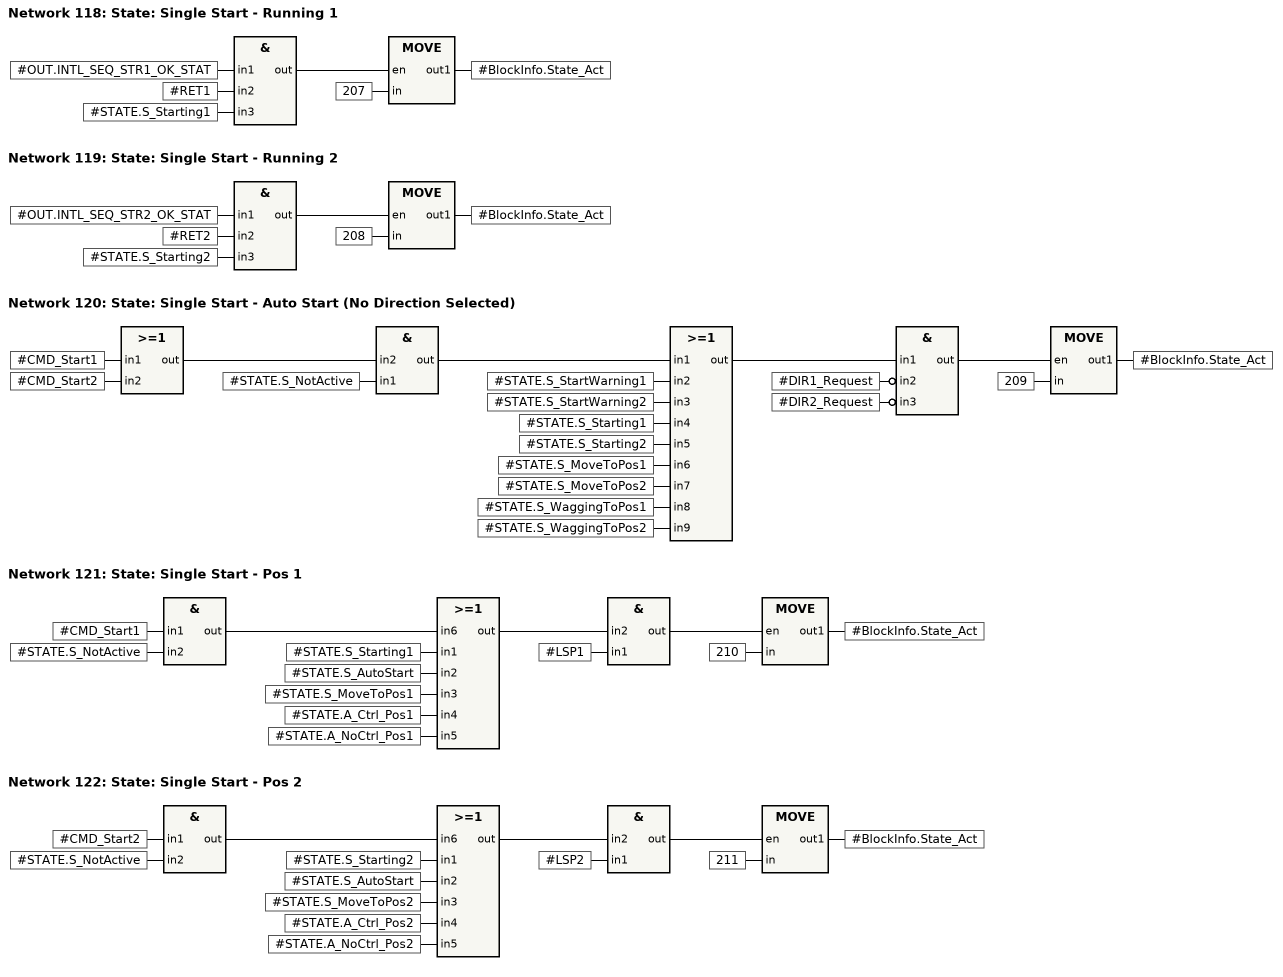
   IF #OUT.INTL_SEQ_STR1_OK_STAT AND #RET1 AND #STATE.S_Starting1 THEN #BlockInfo.State_Act := 207; END_IF;
END_REGION

REGION Network 119: State: Single Start - Running 2
   IF #OUT.INTL_SEQ_STR2_OK_STAT AND #RET2 AND #STATE.S_Starting2 THEN #BlockInfo.State_Act := 208; END_IF;
END_REGION

REGION Network 120: State: Single Start - Auto Start (No Direction Selected)
   IF (((#CMD_Start1 OR #CMD_Start2) AND #STATE.S_NotActive) OR #STATE.S_StartWarning1 OR #STATE.S_StartWarning2 OR #STATE.S_Starting1 OR #STATE.S_Starting2 OR #STATE.S_MoveToPos1 OR #STATE.S_MoveToPos2 OR #STATE.S_WaggingToPos1 OR #STATE.S_WaggingToPos2) AND NOT #DIR1_Request AND NOT #DIR2_Request THEN
       #BlockInfo.State_Act := 209;
   END_IF;
END_REGION

REGION Network 121: State: Single Start - Pos 1
   IF ((#CMD_Start1 AND #STATE.S_NotActive) OR #STATE.S_Starting1 OR #STATE.S_AutoStart OR #STATE.S_MoveToPos1 OR #STATE.A_Ctrl_Pos1 OR #STATE.A_NoCtrl_Pos1) AND #LSP1 THEN
       #BlockInfo.State_Act := 210;
   END_IF;
END_REGION

REGION Network 122: State: Single Start - Pos 2
   IF ((#CMD_Start2 AND #STATE.S_NotActive) OR #STATE.S_Starting2 OR #STATE.S_AutoStart OR #STATE.S_MoveToPos2 OR #STATE.A_Ctrl_Pos2 OR #STATE.A_NoCtrl_Pos2) AND #LSP2 THEN
       #BlockInfo.State_Act := 211;
   END_IF;
END_REGION

REGION Network 123: State: Single Start - Stop
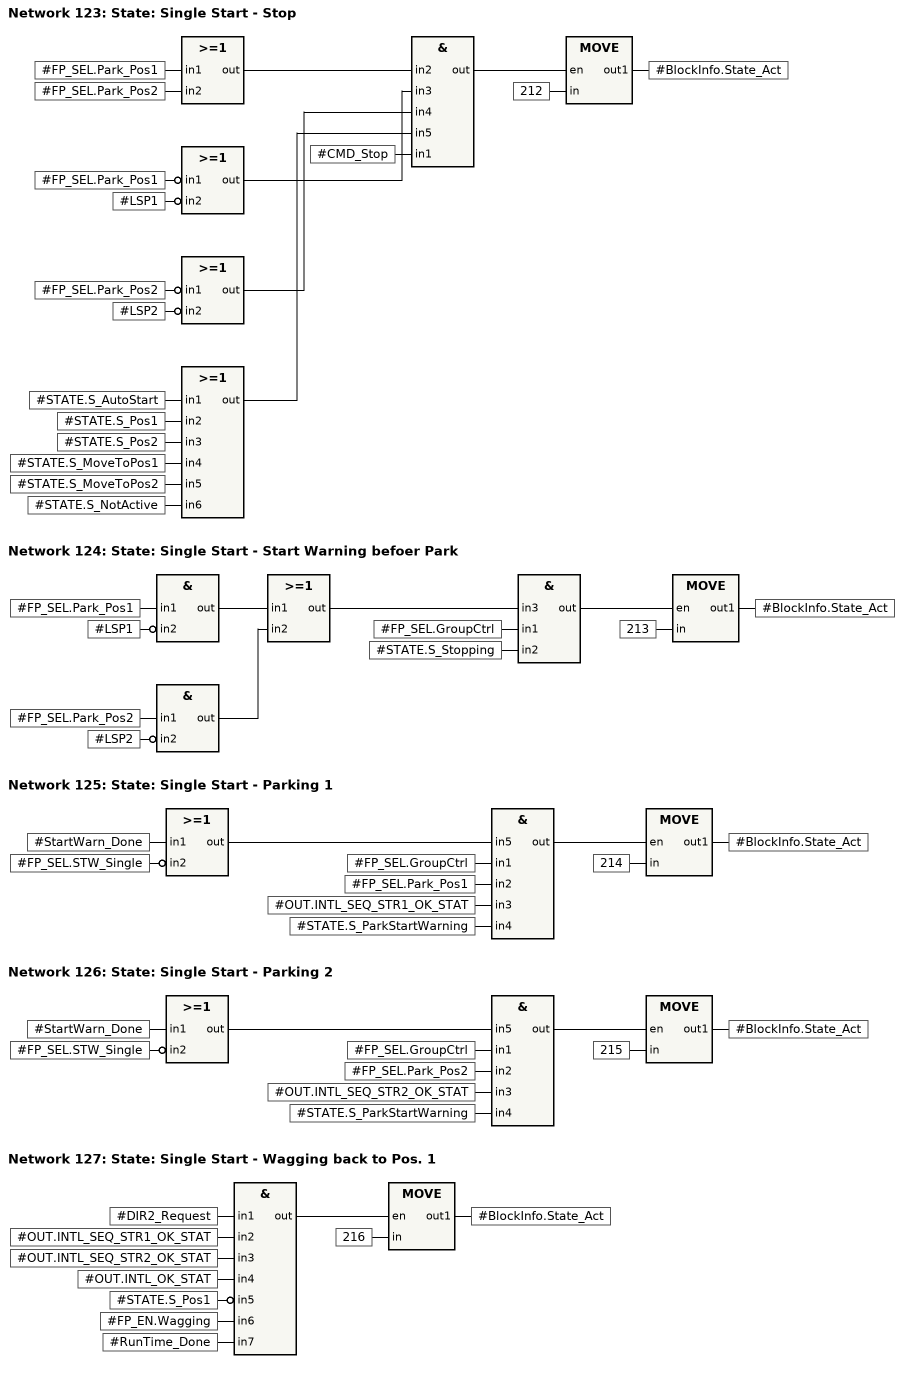
   IF (#FP_SEL.Park_Pos1 OR #FP_SEL.Park_Pos2) AND (NOT #FP_SEL.Park_Pos1 OR NOT #LSP1) AND (NOT #FP_SEL.Park_Pos2 OR NOT #LSP2) AND (#STATE.S_AutoStart OR #STATE.S_Pos1 OR #STATE.S_Pos2 OR #STATE.S_MoveToPos1 OR #STATE.S_MoveToPos2 OR #STATE.S_NotActive) AND #CMD_Stop THEN
       #BlockInfo.State_Act := 212;
   END_IF;
END_REGION

REGION Network 124: State: Single Start - Start Warning befoer Park
   IF ((#FP_SEL.Park_Pos1 AND NOT #LSP1) OR (#FP_SEL.Park_Pos2 AND NOT #LSP2)) AND #FP_SEL.GroupCtrl AND #STATE.S_Stopping THEN
       #BlockInfo.State_Act := 213;
   END_IF;
END_REGION

REGION Network 125: State: Single Start - Parking 1
   IF (#StartWarn_Done OR NOT #FP_SEL.STW_Single) AND #FP_SEL.GroupCtrl AND #FP_SEL.Park_Pos1 AND #OUT.INTL_SEQ_STR1_OK_STAT AND #STATE.S_ParkStartWarning THEN
       #BlockInfo.State_Act := 214;
   END_IF;
END_REGION

REGION Network 126: State: Single Start - Parking 2
   IF (#StartWarn_Done OR NOT #FP_SEL.STW_Single) AND #FP_SEL.GroupCtrl AND #FP_SEL.Park_Pos2 AND #OUT.INTL_SEQ_STR2_OK_STAT AND #STATE.S_ParkStartWarning THEN
       #BlockInfo.State_Act := 215;
   END_IF;
END_REGION

REGION Network 127: State: Single Start - Wagging back to Pos. 1
   IF #DIR2_Request AND #OUT.INTL_SEQ_STR1_OK_STAT AND #OUT.INTL_SEQ_STR2_OK_STAT AND #OUT.INTL_OK_STAT AND NOT #STATE.S_Pos1 AND #FP_EN.Wagging AND #RunTime_Done THEN
       #BlockInfo.State_Act := 216;
   END_IF;
END_REGION

REGION Network 128: State: Single Start - Wagging back to Pos. 2
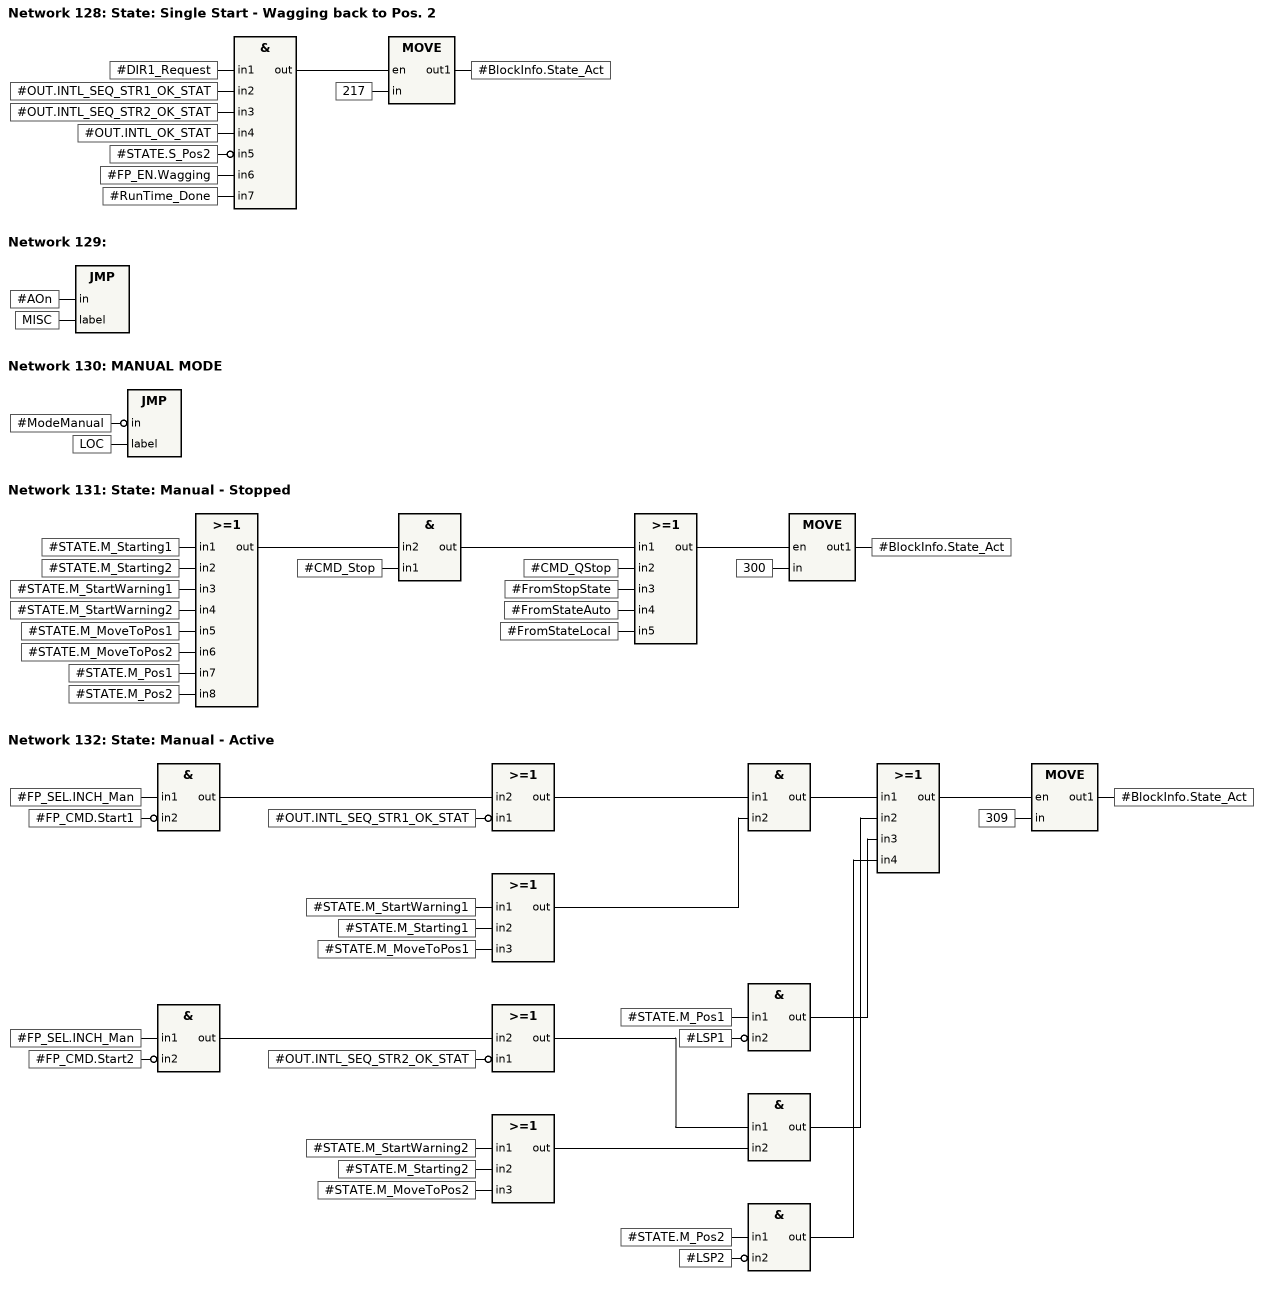
   IF #DIR1_Request AND #OUT.INTL_SEQ_STR1_OK_STAT AND #OUT.INTL_SEQ_STR2_OK_STAT AND #OUT.INTL_OK_STAT AND NOT #STATE.S_Pos2 AND #FP_EN.Wagging AND #RunTime_Done THEN
       #BlockInfo.State_Act := 217;
   END_IF;
END_REGION

REGION Network 129
   IF #AOn THEN GOTO MISC; END_IF;
END_REGION

REGION Network 130: MANUAL MODE
   MAN:
   IF NOT #ModeManual THEN GOTO LOC; END_IF;
END_REGION

REGION Network 131: State: Manual - Stopped
   IF ((#STATE.M_Starting1 OR #STATE.M_Starting2 OR #STATE.M_StartWarning1 OR #STATE.M_StartWarning2 OR #STATE.M_MoveToPos1 OR #STATE.M_MoveToPos2 OR #STATE.M_Pos1 OR #STATE.M_Pos2) AND #CMD_Stop) OR #CMD_QStop OR #FromStopState OR #FromStateAuto OR #FromStateLocal THEN
       #BlockInfo.State_Act := 300;
   END_IF;
END_REGION

REGION Network 132: State: Manual - Active
   // Build 016 - 21.Feb.2022 (SURAM-IN) FP_CMD.Start1,  FP_CMD.Start2 and FP_SEL.INCH_Man logic added for Inching in Manual Mode
   IF (((#FP_SEL.INCH_Man AND NOT #FP_CMD.Start1) OR NOT #OUT.INTL_SEQ_STR1_OK_STAT) AND (#STATE.M_StartWarning1 OR #STATE.M_Starting1 OR #STATE.M_MoveToPos1)) OR (((#FP_SEL.INCH_Man AND NOT #FP_CMD.Start2) OR NOT #OUT.INTL_SEQ_STR2_OK_STAT) AND (#STATE.M_StartWarning2 OR #STATE.M_Starting2 OR #STATE.M_MoveToPos2)) OR (#STATE.M_Pos1 AND NOT #LSP1) OR (#STATE.M_Pos2 AND NOT #LSP2) THEN
       #BlockInfo.State_Act := 309;
   END_IF;
END_REGION

REGION Network 133: State: Manual - Start Warning 1
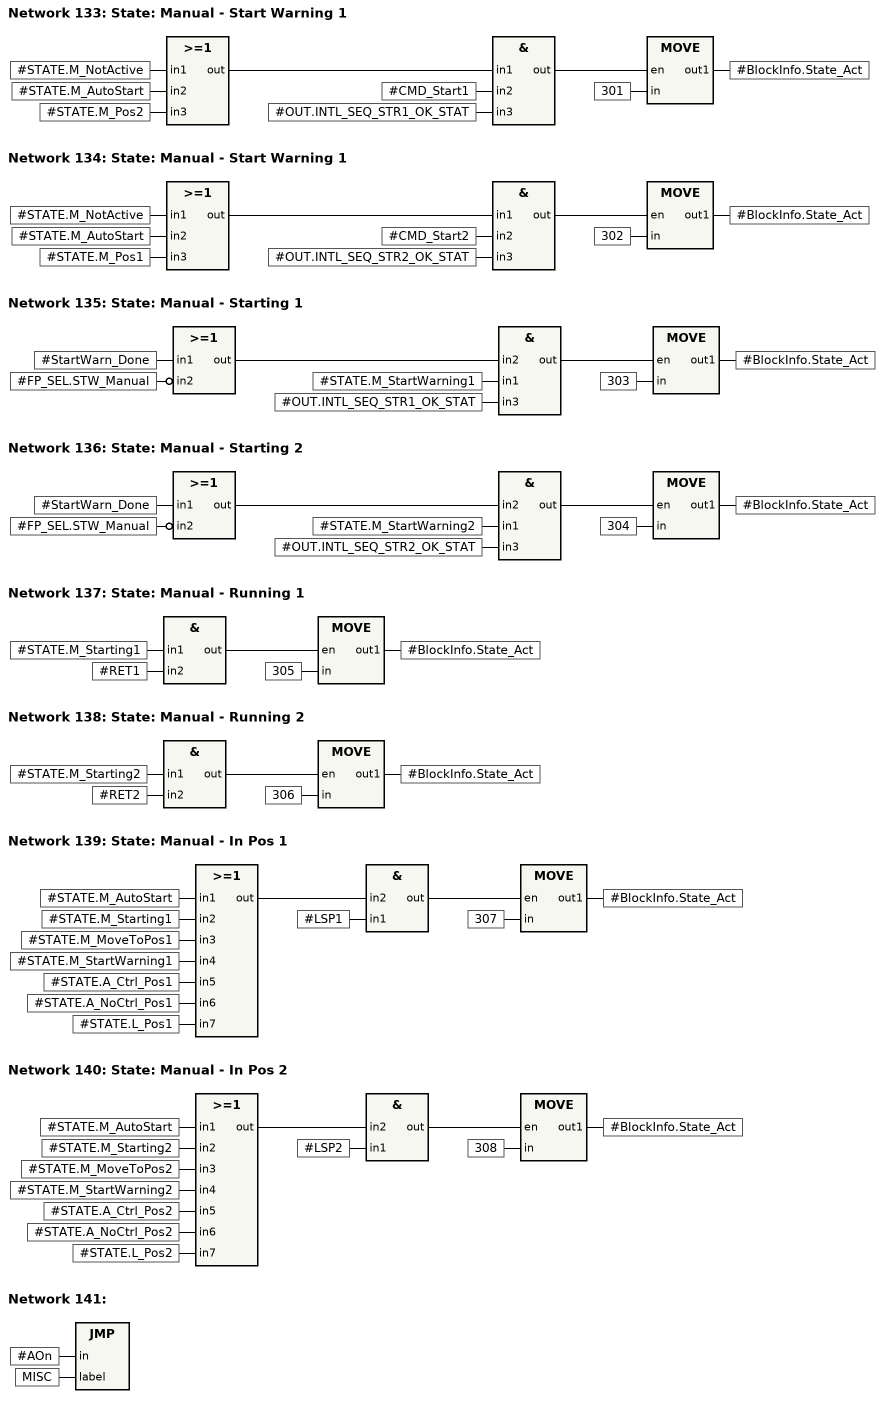
   IF (#STATE.M_NotActive OR #STATE.M_AutoStart OR #STATE.M_Pos2) AND #CMD_Start1 AND #OUT.INTL_SEQ_STR1_OK_STAT THEN
       #BlockInfo.State_Act := 301;
   END_IF;
END_REGION

REGION Network 134: State: Manual - Start Warning 1
   IF (#STATE.M_NotActive OR #STATE.M_AutoStart OR #STATE.M_Pos1) AND #CMD_Start2 AND #OUT.INTL_SEQ_STR2_OK_STAT THEN
       #BlockInfo.State_Act := 302;
   END_IF;
END_REGION

REGION Network 135: State: Manual - Starting 1
   IF (#StartWarn_Done OR NOT #FP_SEL.STW_Manual) AND #STATE.M_StartWarning1 AND #OUT.INTL_SEQ_STR1_OK_STAT THEN
       #BlockInfo.State_Act := 303;
   END_IF;
END_REGION

REGION Network 136: State: Manual - Starting 2
   IF (#StartWarn_Done OR NOT #FP_SEL.STW_Manual) AND #STATE.M_StartWarning2 AND #OUT.INTL_SEQ_STR2_OK_STAT THEN
       #BlockInfo.State_Act := 304;
   END_IF;
END_REGION

REGION Network 137: State: Manual - Running 1
   IF #STATE.M_Starting1 AND #RET1 THEN #BlockInfo.State_Act := 305; END_IF;
END_REGION

REGION Network 138: State: Manual - Running 2
   IF #STATE.M_Starting2 AND #RET2 THEN #BlockInfo.State_Act := 306; END_IF;
END_REGION

REGION Network 139: State: Manual - In Pos 1
   IF (#STATE.M_AutoStart OR #STATE.M_Starting1 OR #STATE.M_MoveToPos1 OR #STATE.M_StartWarning1 OR #STATE.A_Ctrl_Pos1 OR #STATE.A_NoCtrl_Pos1 OR #STATE.L_Pos1) AND #LSP1 THEN
       #BlockInfo.State_Act := 307;
   END_IF;
END_REGION

REGION Network 140: State: Manual - In Pos 2
   IF (#STATE.M_AutoStart OR #STATE.M_Starting2 OR #STATE.M_MoveToPos2 OR #STATE.M_StartWarning2 OR #STATE.A_Ctrl_Pos2 OR #STATE.A_NoCtrl_Pos2 OR #STATE.L_Pos2) AND #LSP2 THEN
       #BlockInfo.State_Act := 308;
   END_IF;
END_REGION

REGION Network 141
   IF #AOn THEN GOTO MISC; END_IF;
END_REGION

REGION Network 142: LOCAL MODE
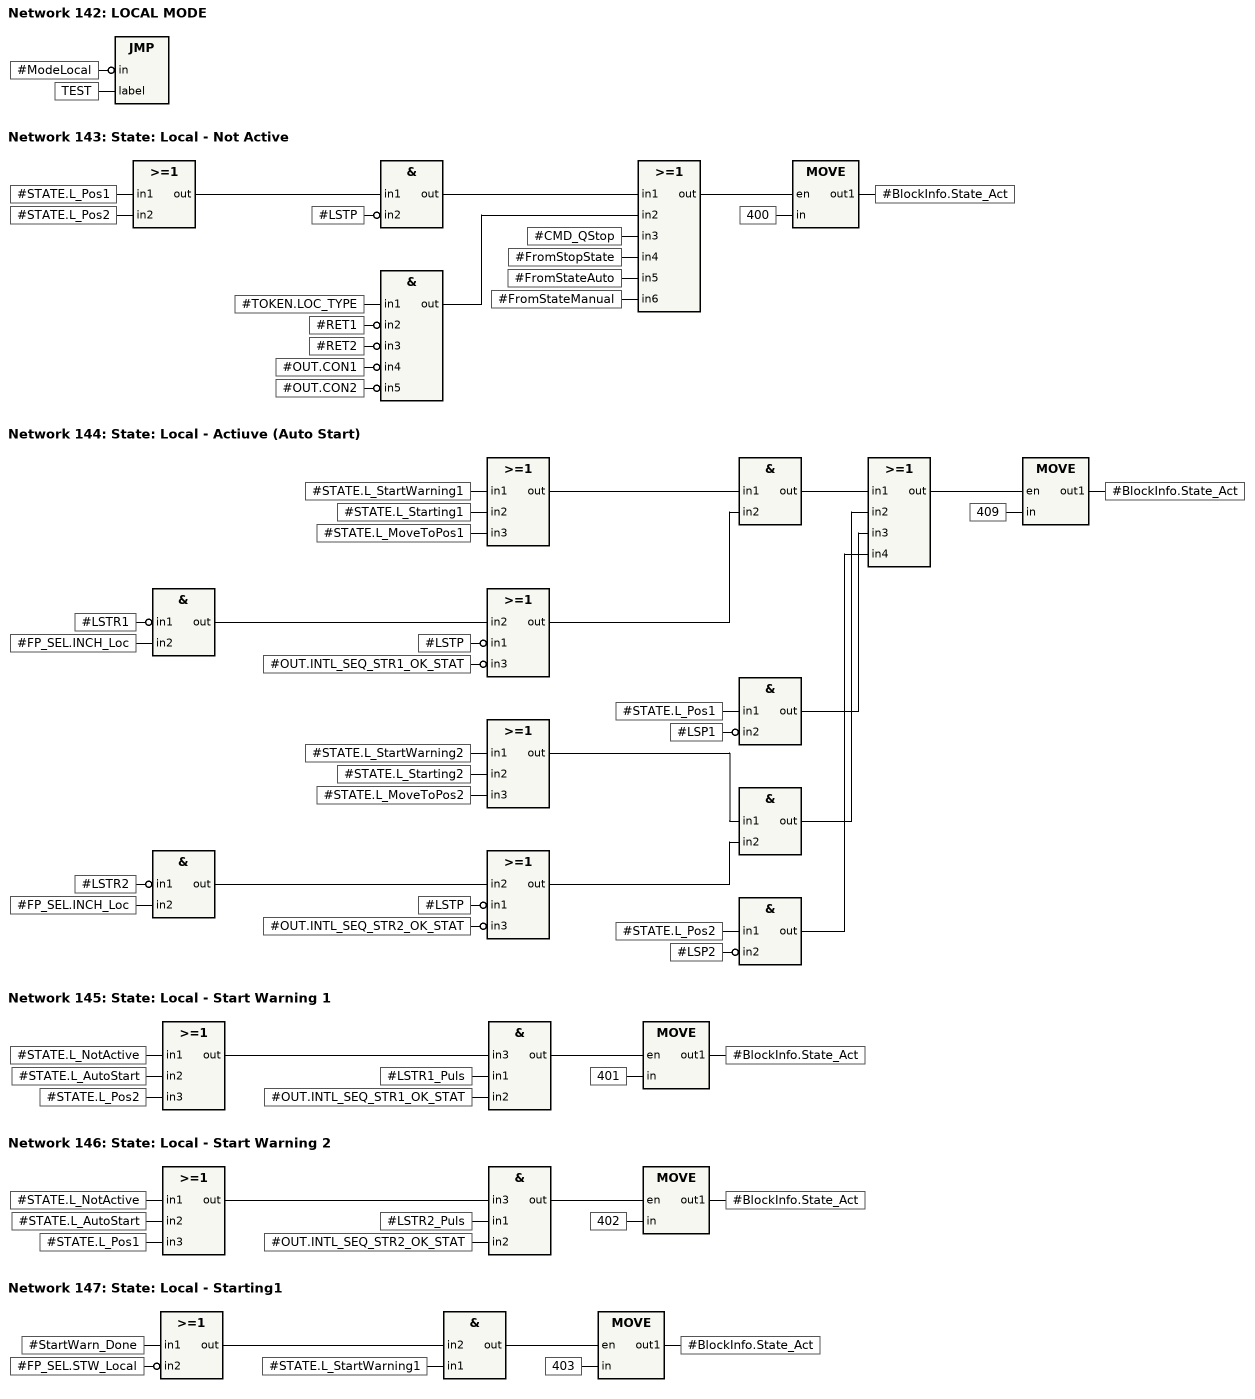
   LOC:
   IF NOT #ModeLocal THEN GOTO TEST; END_IF;
END_REGION

REGION Network 143: State: Local - Not Active
   IF ((#STATE.L_Pos1 OR #STATE.L_Pos2) AND NOT #LSTP) OR (#TOKEN.LOC_TYPE AND NOT #RET1 AND NOT #RET2 AND NOT #OUT.CON1 AND NOT #OUT.CON2) OR #CMD_QStop OR #FromStopState OR #FromStateAuto OR #FromStateManual THEN
       #BlockInfo.State_Act := 400;
   END_IF;
END_REGION

REGION Network 144: State: Local - Actiuve (Auto Start)
   IF ((#STATE.L_StartWarning1 OR #STATE.L_Starting1 OR #STATE.L_MoveToPos1) AND ((NOT #LSTR1 AND #FP_SEL.INCH_Loc) OR NOT #LSTP OR NOT #OUT.INTL_SEQ_STR1_OK_STAT)) OR ((#STATE.L_StartWarning2 OR #STATE.L_Starting2 OR #STATE.L_MoveToPos2) AND ((NOT #LSTR2 AND #FP_SEL.INCH_Loc) OR NOT #LSTP OR NOT #OUT.INTL_SEQ_STR2_OK_STAT)) OR (#STATE.L_Pos1 AND NOT #LSP1) OR (#STATE.L_Pos2 AND NOT #LSP2) THEN
       #BlockInfo.State_Act := 409;
   END_IF;
END_REGION

REGION Network 145: State: Local - Start Warning 1
   IF (#STATE.L_NotActive OR #STATE.L_AutoStart OR #STATE.L_Pos2) AND #LSTR1_Puls AND #OUT.INTL_SEQ_STR1_OK_STAT THEN
       #BlockInfo.State_Act := 401;
   END_IF;
END_REGION

REGION Network 146: State: Local - Start Warning 2
   IF (#STATE.L_NotActive OR #STATE.L_AutoStart OR #STATE.L_Pos1) AND #LSTR2_Puls AND #OUT.INTL_SEQ_STR2_OK_STAT THEN
       #BlockInfo.State_Act := 402;
   END_IF;
END_REGION

REGION Network 147: State: Local - Starting1
   IF (#StartWarn_Done OR NOT #FP_SEL.STW_Local) AND #STATE.L_StartWarning1 THEN
       #BlockInfo.State_Act := 403;
   END_IF;
END_REGION

REGION Network 148: State: Local - Starting2
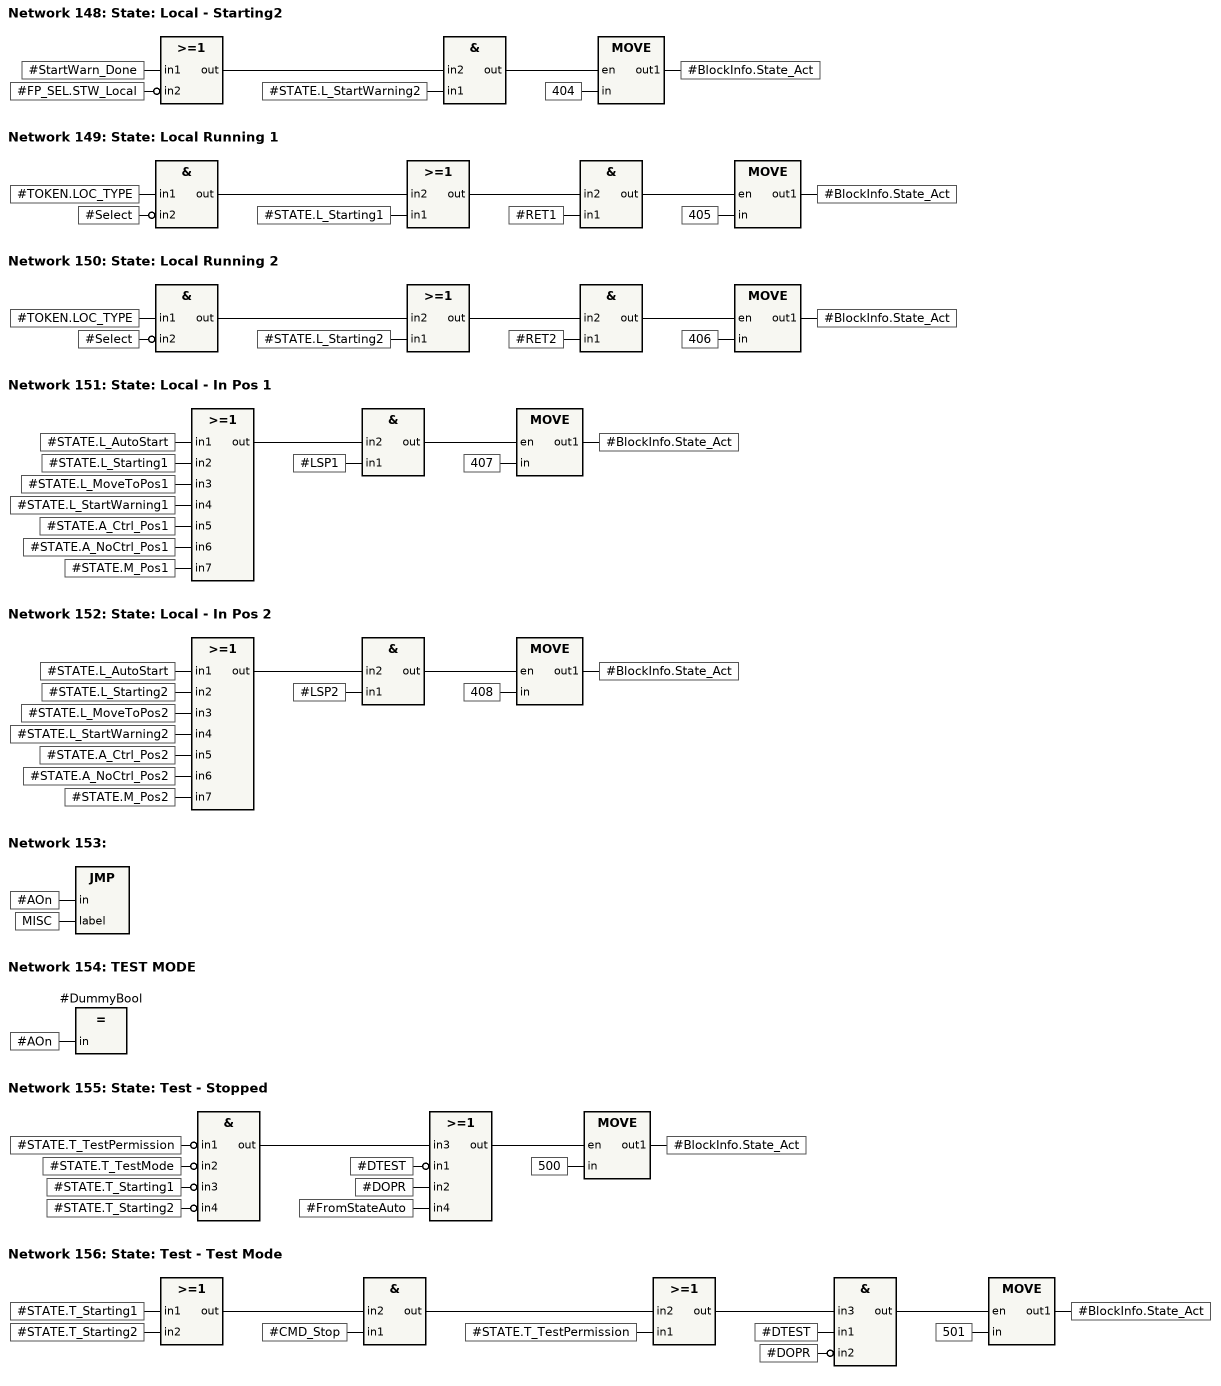
   IF (#StartWarn_Done OR NOT #FP_SEL.STW_Local) AND #STATE.L_StartWarning2 THEN
       #BlockInfo.State_Act := 404;
   END_IF;
END_REGION

REGION Network 149: State: Local Running 1
   IF ((#TOKEN.LOC_TYPE AND NOT #Select) OR #STATE.L_Starting1) AND #RET1 THEN
       #BlockInfo.State_Act := 405;
   END_IF;
END_REGION

REGION Network 150: State: Local Running 2
   IF ((#TOKEN.LOC_TYPE AND NOT #Select) OR #STATE.L_Starting2) AND #RET2 THEN
       #BlockInfo.State_Act := 406;
   END_IF;
END_REGION

REGION Network 151: State: Local - In Pos 1
   IF (#STATE.L_AutoStart OR #STATE.L_Starting1 OR #STATE.L_MoveToPos1 OR #STATE.L_StartWarning1 OR #STATE.A_Ctrl_Pos1 OR #STATE.A_NoCtrl_Pos1 OR #STATE.M_Pos1) AND #LSP1 THEN
       #BlockInfo.State_Act := 407;
   END_IF;
END_REGION

REGION Network 152: State: Local - In Pos 2
   IF (#STATE.L_AutoStart OR #STATE.L_Starting2 OR #STATE.L_MoveToPos2 OR #STATE.L_StartWarning2 OR #STATE.A_Ctrl_Pos2 OR #STATE.A_NoCtrl_Pos2 OR #STATE.M_Pos2) AND #LSP2 THEN
       #BlockInfo.State_Act := 408;
   END_IF;
END_REGION

REGION Network 153
   IF #AOn THEN GOTO MISC; END_IF;
END_REGION

REGION Network 154: TEST MODE
   TEST:
   #DummyBool := #AOn;
END_REGION

REGION Network 155: State: Test - Stopped
   IF (NOT #STATE.T_TestPermission AND NOT #STATE.T_TestMode AND NOT #STATE.T_Starting1 AND NOT #STATE.T_Starting2) OR NOT #DTEST OR #DOPR OR #FromStateAuto THEN
       #BlockInfo.State_Act := 500;
   END_IF;
END_REGION

REGION Network 156: State: Test - Test Mode
   IF (((#STATE.T_Starting1 OR #STATE.T_Starting2) AND #CMD_Stop) OR #STATE.T_TestPermission) AND #DTEST AND NOT #DOPR THEN
       #BlockInfo.State_Act := 501;
   END_IF;
END_REGION

REGION Network 157: State: Test - Starting 1
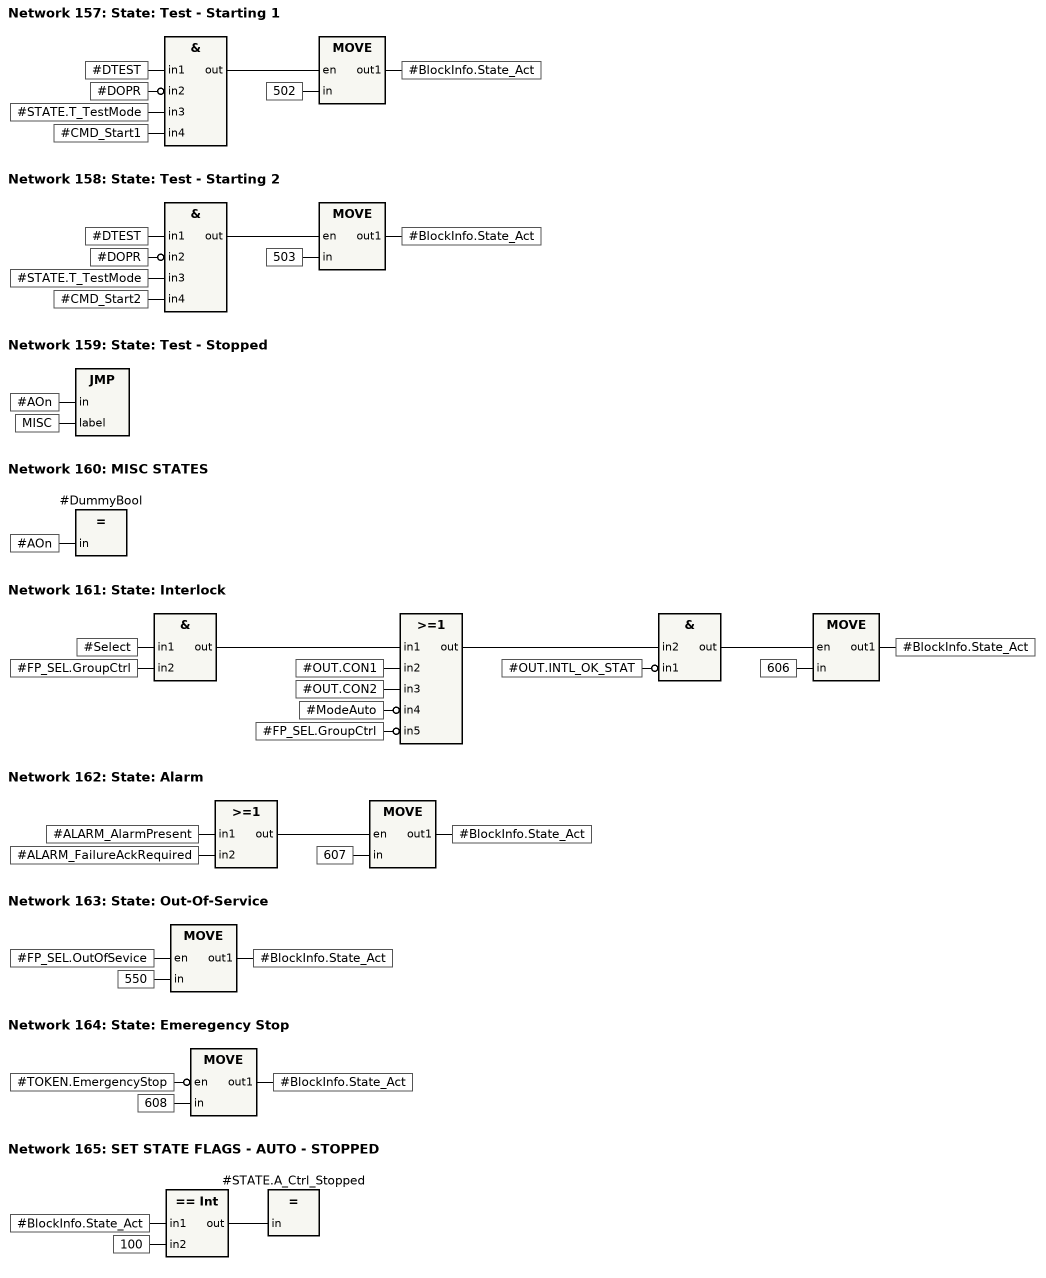
   IF #DTEST AND NOT #DOPR AND #STATE.T_TestMode AND #CMD_Start1 THEN #BlockInfo.State_Act := 502; END_IF;
END_REGION

REGION Network 158: State: Test - Starting 2
   IF #DTEST AND NOT #DOPR AND #STATE.T_TestMode AND #CMD_Start2 THEN #BlockInfo.State_Act := 503; END_IF;
END_REGION

REGION Network 159: State: Test - Stopped
   IF #AOn THEN GOTO MISC; END_IF;
END_REGION

REGION Network 160: MISC STATES
   MISC:
   #DummyBool := #AOn;
END_REGION

REGION Network 161: State: Interlock
   IF ((#Select AND #FP_SEL.GroupCtrl) OR #OUT.CON1 OR #OUT.CON2 OR NOT #ModeAuto OR NOT #FP_SEL.GroupCtrl) AND NOT #OUT.INTL_OK_STAT THEN
       #BlockInfo.State_Act := 606;
   END_IF;
END_REGION

REGION Network 162: State: Alarm
   IF #ALARM_AlarmPresent OR #ALARM_FailureAckRequired THEN #BlockInfo.State_Act := 607; END_IF;
END_REGION

REGION Network 163: State: Out-Of-Service
   IF #FP_SEL.OutOfSevice THEN #BlockInfo.State_Act := 550; END_IF;
END_REGION

REGION Network 164: State: Emeregency Stop
   IF NOT #TOKEN.EmergencyStop THEN #BlockInfo.State_Act := 608; END_IF;
END_REGION

REGION Network 165: SET STATE FLAGS - AUTO - STOPPED
   #STATE.A_Ctrl_Stopped := #BlockInfo.State_Act = 100;
END_REGION

REGION Network 166: SET STATE FLAGS - AUTO - SELECTED
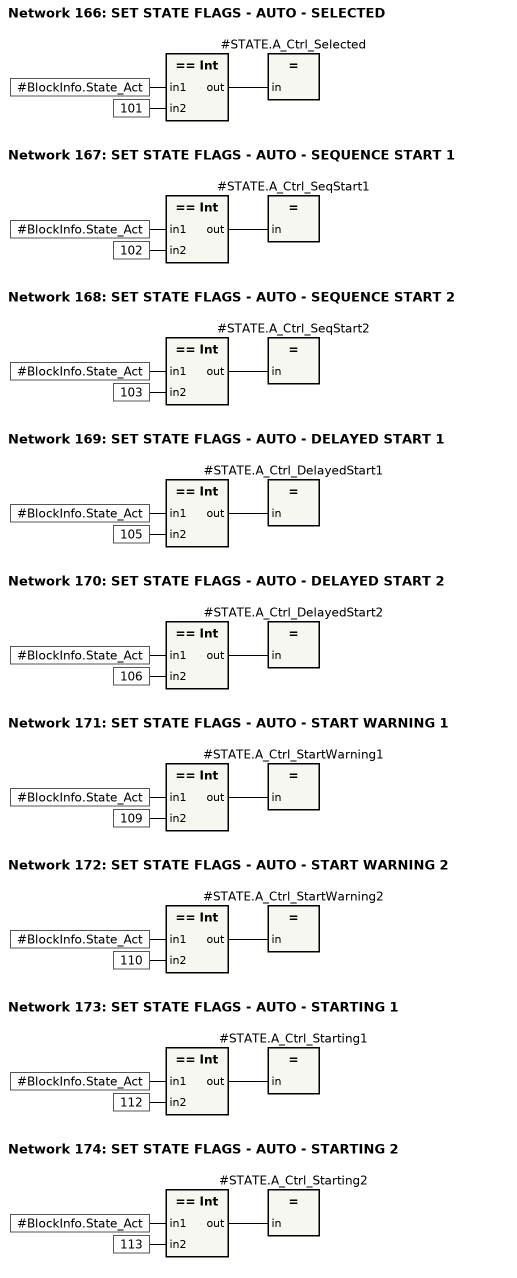
   #STATE.A_Ctrl_Selected := #BlockInfo.State_Act = 101;
END_REGION

REGION Network 167: SET STATE FLAGS - AUTO - SEQUENCE START 1
   #STATE.A_Ctrl_SeqStart1 := #BlockInfo.State_Act = 102;
END_REGION

REGION Network 168: SET STATE FLAGS - AUTO - SEQUENCE START 2
   #STATE.A_Ctrl_SeqStart2 := #BlockInfo.State_Act = 103;
END_REGION

REGION Network 169: SET STATE FLAGS - AUTO - DELAYED START 1
   #STATE.A_Ctrl_DelayedStart1 := #BlockInfo.State_Act = 105;
END_REGION

REGION Network 170: SET STATE FLAGS - AUTO - DELAYED START 2
   #STATE.A_Ctrl_DelayedStart2 := #BlockInfo.State_Act = 106;
END_REGION

REGION Network 171: SET STATE FLAGS - AUTO - START WARNING 1
   #STATE.A_Ctrl_StartWarning1 := #BlockInfo.State_Act = 109;
END_REGION

REGION Network 172: SET STATE FLAGS - AUTO - START WARNING 2
   #STATE.A_Ctrl_StartWarning2 := #BlockInfo.State_Act = 110;
END_REGION

REGION Network 173: SET STATE FLAGS - AUTO - STARTING 1
   #STATE.A_Ctrl_Starting1 := #BlockInfo.State_Act = 112;
END_REGION

REGION Network 174: SET STATE FLAGS - AUTO - STARTING 2
   #STATE.A_Ctrl_Starting2 := #BlockInfo.State_Act = 113;
END_REGION

REGION Network 175: SET STATE FLAGS - AUTO - MOVE TO POS 1
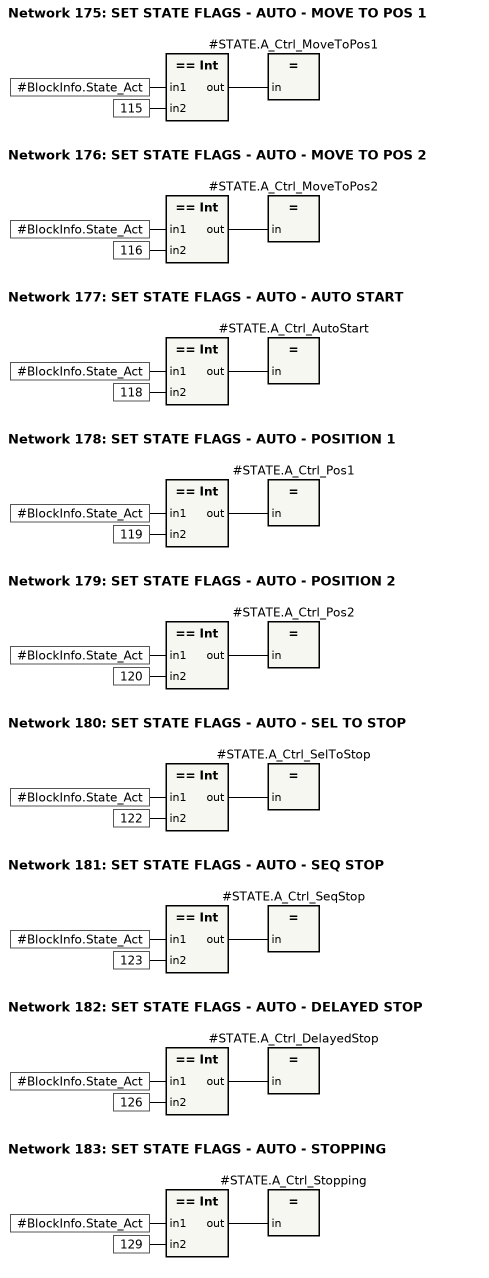
   #STATE.A_Ctrl_MoveToPos1 := #BlockInfo.State_Act = 115;
END_REGION

REGION Network 176: SET STATE FLAGS - AUTO - MOVE TO POS 2
   #STATE.A_Ctrl_MoveToPos2 := #BlockInfo.State_Act = 116;
END_REGION

REGION Network 177: SET STATE FLAGS - AUTO - AUTO START
   #STATE.A_Ctrl_AutoStart := #BlockInfo.State_Act = 118;
END_REGION

REGION Network 178: SET STATE FLAGS - AUTO - POSITION 1
   #STATE.A_Ctrl_Pos1 := #BlockInfo.State_Act = 119;
END_REGION

REGION Network 179: SET STATE FLAGS - AUTO - POSITION 2
   #STATE.A_Ctrl_Pos2 := #BlockInfo.State_Act = 120;
END_REGION

REGION Network 180: SET STATE FLAGS - AUTO - SEL TO STOP
   #STATE.A_Ctrl_SelToStop := #BlockInfo.State_Act = 122;
END_REGION

REGION Network 181: SET STATE FLAGS - AUTO - SEQ STOP
   #STATE.A_Ctrl_SeqStop := #BlockInfo.State_Act = 123;
END_REGION

REGION Network 182: SET STATE FLAGS - AUTO - DELAYED STOP
   #STATE.A_Ctrl_DelayedStop := #BlockInfo.State_Act = 126;
END_REGION

REGION Network 183: SET STATE FLAGS - AUTO - STOPPING
   #STATE.A_Ctrl_Stopping := #BlockInfo.State_Act = 129;
END_REGION

REGION Network 184: SET STATE FLAGS - AUTO - PARK START WARNING
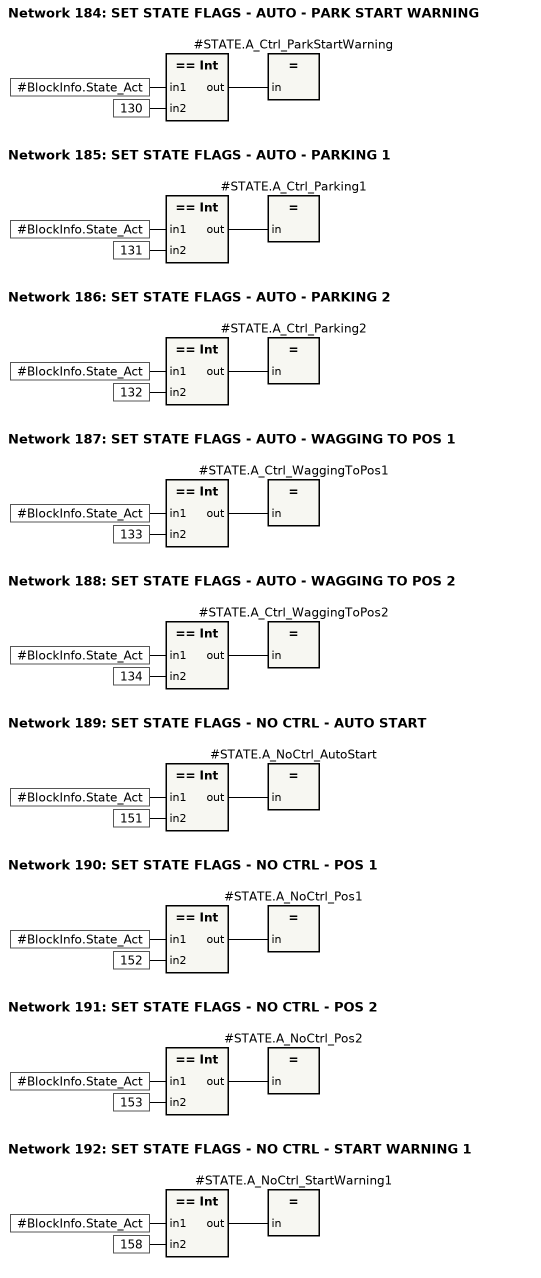
   #STATE.A_Ctrl_ParkStartWarning := #BlockInfo.State_Act = 130;
END_REGION

REGION Network 185: SET STATE FLAGS - AUTO - PARKING 1
   #STATE.A_Ctrl_Parking1 := #BlockInfo.State_Act = 131;
END_REGION

REGION Network 186: SET STATE FLAGS - AUTO - PARKING 2
   #STATE.A_Ctrl_Parking2 := #BlockInfo.State_Act = 132;
END_REGION

REGION Network 187: SET STATE FLAGS - AUTO - WAGGING TO POS 1
   #STATE.A_Ctrl_WaggingToPos1 := #BlockInfo.State_Act = 133;
END_REGION

REGION Network 188: SET STATE FLAGS - AUTO - WAGGING TO POS 2
   #STATE.A_Ctrl_WaggingToPos2 := #BlockInfo.State_Act = 134;
END_REGION

REGION Network 189: SET STATE FLAGS - NO CTRL - AUTO START
   #STATE.A_NoCtrl_AutoStart := #BlockInfo.State_Act = 151;
END_REGION

REGION Network 190: SET STATE FLAGS - NO CTRL - POS 1
   #STATE.A_NoCtrl_Pos1 := #BlockInfo.State_Act = 152;
END_REGION

REGION Network 191: SET STATE FLAGS - NO CTRL - POS 2
   #STATE.A_NoCtrl_Pos2 := #BlockInfo.State_Act = 153;
END_REGION

REGION Network 192: SET STATE FLAGS - NO CTRL - START WARNING 1
   #STATE.A_NoCtrl_StartWarning1 := #BlockInfo.State_Act = 158;
END_REGION

REGION Network 193: SET STATE FLAGS - NO CTRL - START WARNING 2
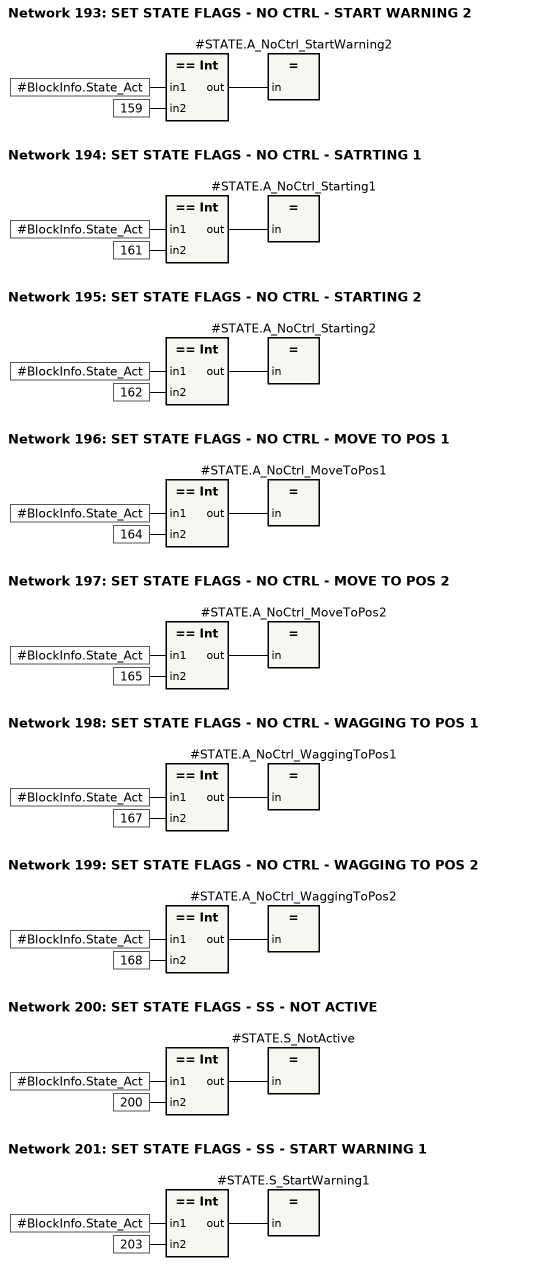
   #STATE.A_NoCtrl_StartWarning2 := #BlockInfo.State_Act = 159;
END_REGION

REGION Network 194: SET STATE FLAGS - NO CTRL - SATRTING 1
   #STATE.A_NoCtrl_Starting1 := #BlockInfo.State_Act = 161;
END_REGION

REGION Network 195: SET STATE FLAGS - NO CTRL - STARTING 2
   #STATE.A_NoCtrl_Starting2 := #BlockInfo.State_Act = 162;
END_REGION

REGION Network 196: SET STATE FLAGS - NO CTRL - MOVE TO POS 1
   #STATE.A_NoCtrl_MoveToPos1 := #BlockInfo.State_Act = 164;
END_REGION

REGION Network 197: SET STATE FLAGS - NO CTRL - MOVE TO POS 2
   #STATE.A_NoCtrl_MoveToPos2 := #BlockInfo.State_Act = 165;
END_REGION

REGION Network 198: SET STATE FLAGS - NO CTRL - WAGGING TO POS 1
   #STATE.A_NoCtrl_WaggingToPos1 := #BlockInfo.State_Act = 167;
END_REGION

REGION Network 199: SET STATE FLAGS - NO CTRL - WAGGING TO POS 2
   #STATE.A_NoCtrl_WaggingToPos2 := #BlockInfo.State_Act = 168;
END_REGION

REGION Network 200: SET STATE FLAGS - SS - NOT ACTIVE
   #STATE.S_NotActive := #BlockInfo.State_Act = 200;
END_REGION

REGION Network 201: SET STATE FLAGS - SS - START WARNING 1
   #STATE.S_StartWarning1 := #BlockInfo.State_Act = 203;
END_REGION

REGION Network 202: SET STATE FLAGS - SS - START WARNING 2
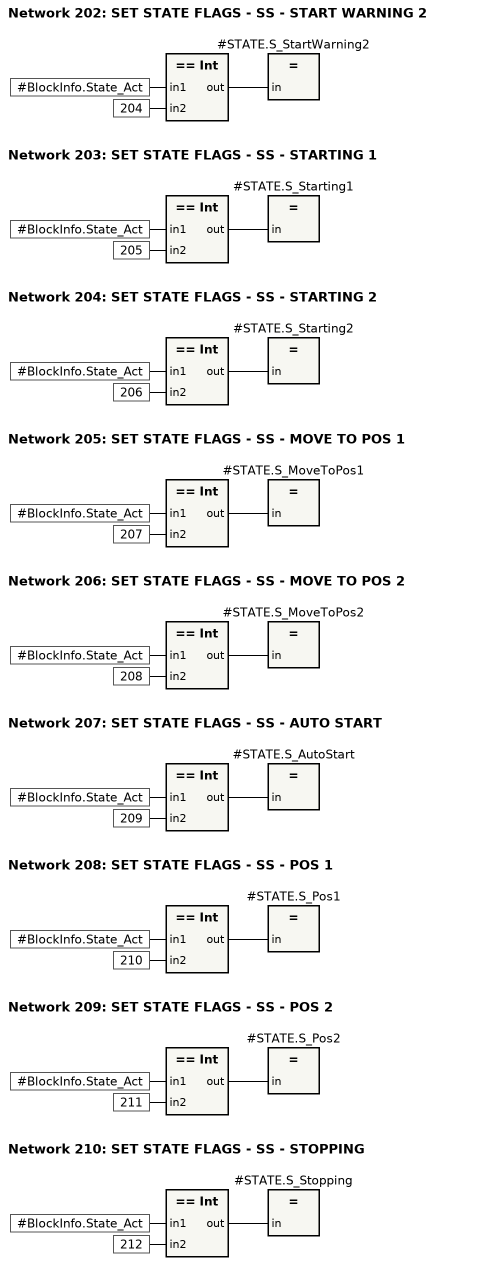
   #STATE.S_StartWarning2 := #BlockInfo.State_Act = 204;
END_REGION

REGION Network 203: SET STATE FLAGS - SS - STARTING 1
   #STATE.S_Starting1 := #BlockInfo.State_Act = 205;
END_REGION

REGION Network 204: SET STATE FLAGS - SS - STARTING 2
   #STATE.S_Starting2 := #BlockInfo.State_Act = 206;
END_REGION

REGION Network 205: SET STATE FLAGS - SS - MOVE TO POS 1
   #STATE.S_MoveToPos1 := #BlockInfo.State_Act = 207;
END_REGION

REGION Network 206: SET STATE FLAGS - SS - MOVE TO POS 2
   #STATE.S_MoveToPos2 := #BlockInfo.State_Act = 208;
END_REGION

REGION Network 207: SET STATE FLAGS - SS - AUTO START
   #STATE.S_AutoStart := #BlockInfo.State_Act = 209;
END_REGION

REGION Network 208: SET STATE FLAGS - SS - POS 1
   #STATE.S_Pos1 := #BlockInfo.State_Act = 210;
END_REGION

REGION Network 209: SET STATE FLAGS - SS - POS 2
   #STATE.S_Pos2 := #BlockInfo.State_Act = 211;
END_REGION

REGION Network 210: SET STATE FLAGS - SS - STOPPING
   #STATE.S_Stopping := #BlockInfo.State_Act = 212;
END_REGION

REGION Network 211: SET STATE FLAGS - SS - PARK START WARNING
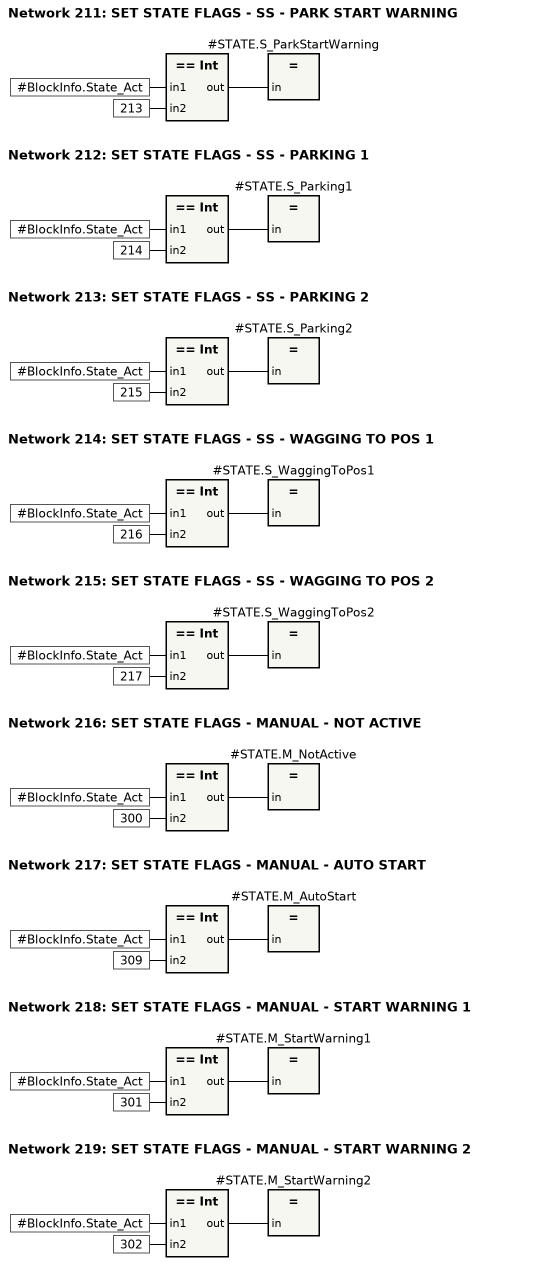
   #STATE.S_ParkStartWarning := #BlockInfo.State_Act = 213;
END_REGION

REGION Network 212: SET STATE FLAGS - SS - PARKING 1
   #STATE.S_Parking1 := #BlockInfo.State_Act = 214;
END_REGION

REGION Network 213: SET STATE FLAGS - SS - PARKING 2
   #STATE.S_Parking2 := #BlockInfo.State_Act = 215;
END_REGION

REGION Network 214: SET STATE FLAGS - SS - WAGGING TO POS 1
   #STATE.S_WaggingToPos1 := #BlockInfo.State_Act = 216;
END_REGION

REGION Network 215: SET STATE FLAGS - SS - WAGGING TO POS 2
   #STATE.S_WaggingToPos2 := #BlockInfo.State_Act = 217;
END_REGION

REGION Network 216: SET STATE FLAGS - MANUAL - NOT ACTIVE
   #STATE.M_NotActive := #BlockInfo.State_Act = 300;
END_REGION

REGION Network 217: SET STATE FLAGS - MANUAL - AUTO START
   #STATE.M_AutoStart := #BlockInfo.State_Act = 309;
END_REGION

REGION Network 218: SET STATE FLAGS - MANUAL - START WARNING 1
   #STATE.M_StartWarning1 := #BlockInfo.State_Act = 301;
END_REGION

REGION Network 219: SET STATE FLAGS - MANUAL - START WARNING 2
   #STATE.M_StartWarning2 := #BlockInfo.State_Act = 302;
END_REGION

REGION Network 220: SET STATE FLAGS - MANUAL - STARTING 1
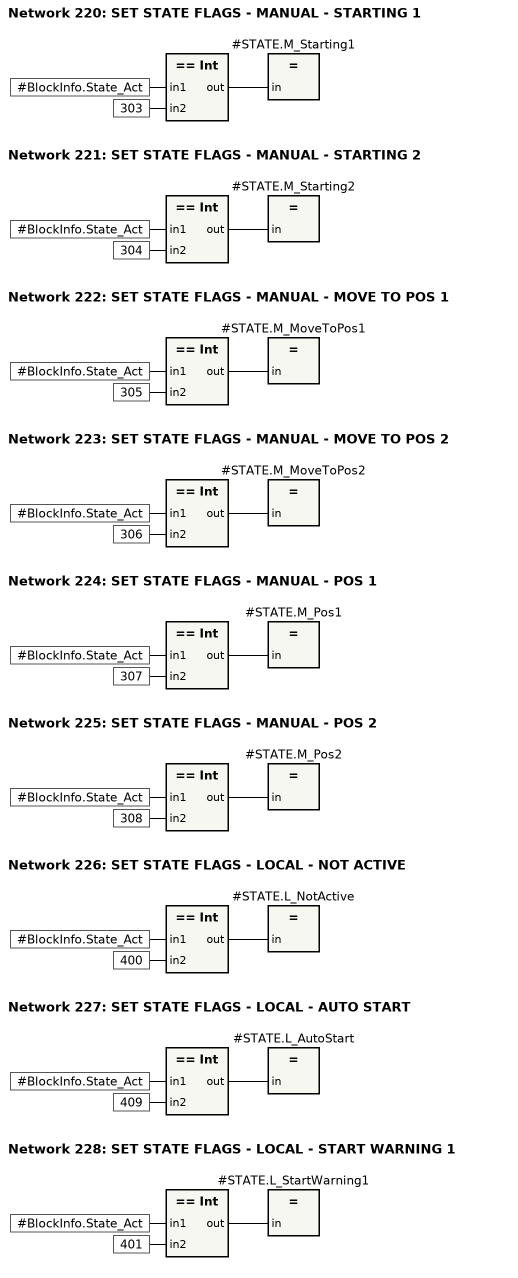
   #STATE.M_Starting1 := #BlockInfo.State_Act = 303;
END_REGION

REGION Network 221: SET STATE FLAGS - MANUAL - STARTING 2
   #STATE.M_Starting2 := #BlockInfo.State_Act = 304;
END_REGION

REGION Network 222: SET STATE FLAGS - MANUAL - MOVE TO POS 1
   #STATE.M_MoveToPos1 := #BlockInfo.State_Act = 305;
END_REGION

REGION Network 223: SET STATE FLAGS - MANUAL - MOVE TO POS 2
   #STATE.M_MoveToPos2 := #BlockInfo.State_Act = 306;
END_REGION

REGION Network 224: SET STATE FLAGS - MANUAL - POS 1
   #STATE.M_Pos1 := #BlockInfo.State_Act = 307;
END_REGION

REGION Network 225: SET STATE FLAGS - MANUAL - POS 2
   #STATE.M_Pos2 := #BlockInfo.State_Act = 308;
END_REGION

REGION Network 226: SET STATE FLAGS - LOCAL - NOT ACTIVE
   #STATE.L_NotActive := #BlockInfo.State_Act = 400;
END_REGION

REGION Network 227: SET STATE FLAGS - LOCAL - AUTO START
   #STATE.L_AutoStart := #BlockInfo.State_Act = 409;
END_REGION

REGION Network 228: SET STATE FLAGS - LOCAL - START WARNING 1
   #STATE.L_StartWarning1 := #BlockInfo.State_Act = 401;
END_REGION

REGION Network 229: SET STATE FLAGS - LOCAL - START WARNING 2
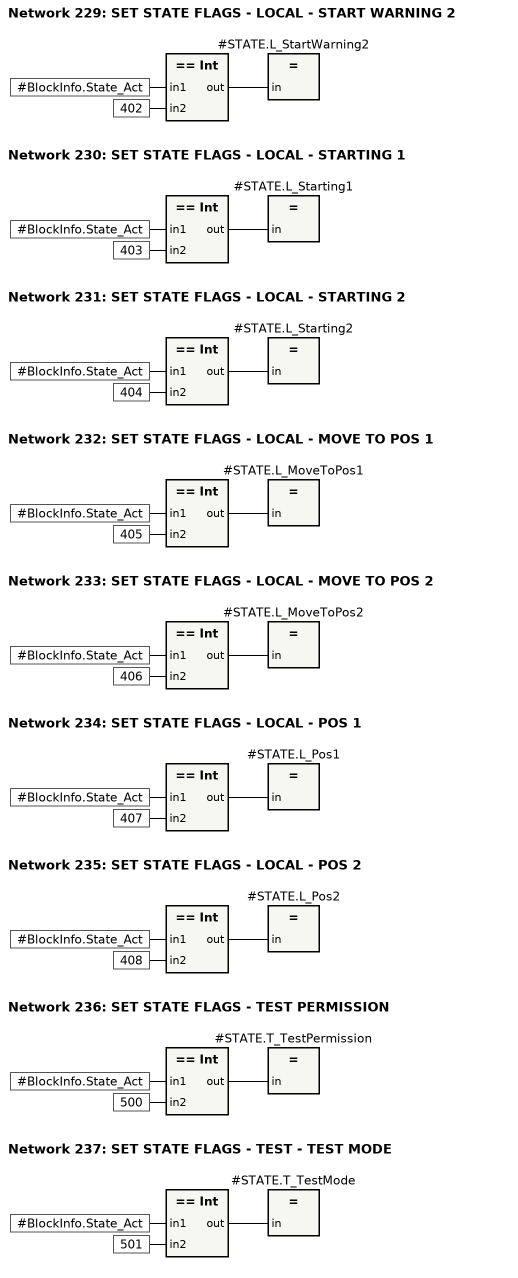
   #STATE.L_StartWarning2 := #BlockInfo.State_Act = 402;
END_REGION

REGION Network 230: SET STATE FLAGS - LOCAL - STARTING 1
   #STATE.L_Starting1 := #BlockInfo.State_Act = 403;
END_REGION

REGION Network 231: SET STATE FLAGS - LOCAL - STARTING 2
   #STATE.L_Starting2 := #BlockInfo.State_Act = 404;
END_REGION

REGION Network 232: SET STATE FLAGS - LOCAL - MOVE TO POS 1
   #STATE.L_MoveToPos1 := #BlockInfo.State_Act = 405;
END_REGION

REGION Network 233: SET STATE FLAGS - LOCAL - MOVE TO POS 2
   #STATE.L_MoveToPos2 := #BlockInfo.State_Act = 406;
END_REGION

REGION Network 234: SET STATE FLAGS - LOCAL - POS 1
   #STATE.L_Pos1 := #BlockInfo.State_Act = 407;
END_REGION

REGION Network 235: SET STATE FLAGS - LOCAL - POS 2
   #STATE.L_Pos2 := #BlockInfo.State_Act = 408;
END_REGION

REGION Network 236: SET STATE FLAGS - TEST PERMISSION
   #STATE.T_TestPermission := #BlockInfo.State_Act = 500;
END_REGION

REGION Network 237: SET STATE FLAGS - TEST - TEST MODE
   #STATE.T_TestMode := #BlockInfo.State_Act = 501;
END_REGION

REGION Network 238: SET STATE FLAGS - TEST - STARTING 1
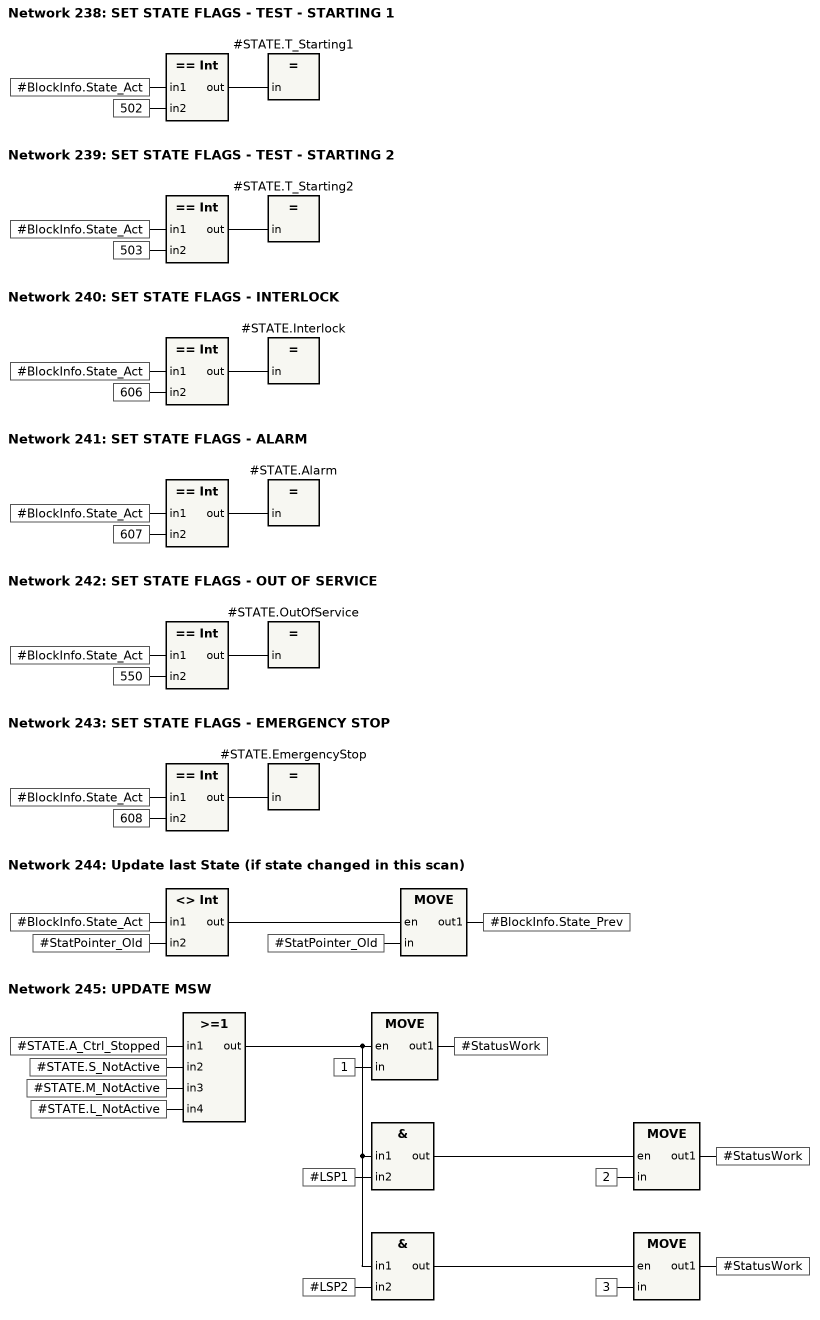
   #STATE.T_Starting1 := #BlockInfo.State_Act = 502;
END_REGION

REGION Network 239: SET STATE FLAGS - TEST - STARTING 2
   #STATE.T_Starting2 := #BlockInfo.State_Act = 503;
END_REGION

REGION Network 240: SET STATE FLAGS - INTERLOCK
   #STATE.Interlock := #BlockInfo.State_Act = 606;
END_REGION

REGION Network 241: SET STATE FLAGS - ALARM
   #STATE.Alarm := #BlockInfo.State_Act = 607;
END_REGION

REGION Network 242: SET STATE FLAGS - OUT OF SERVICE
   #STATE.OutOfService := #BlockInfo.State_Act = 550;
END_REGION

REGION Network 243: SET STATE FLAGS - EMERGENCY STOP
   #STATE.EmergencyStop := #BlockInfo.State_Act = 608;
END_REGION

REGION Network 244: Update last State (if state changed in this scan)
   IF #BlockInfo.State_Act <> #StatPointer_Old THEN #BlockInfo.State_Prev := #StatPointer_Old; END_IF;
END_REGION

REGION Network 245: UPDATE MSW
   #_w1 := #STATE.A_Ctrl_Stopped OR #STATE.S_NotActive OR #STATE.M_NotActive OR #STATE.L_NotActive;
   IF #_w1 THEN #StatusWork := 1; END_IF;
   IF #_w1 AND #LSP1 THEN #StatusWork := 2; END_IF;
   IF #_w1 AND #LSP2 THEN #StatusWork := 3; END_IF;
END_REGION

REGION Network 246
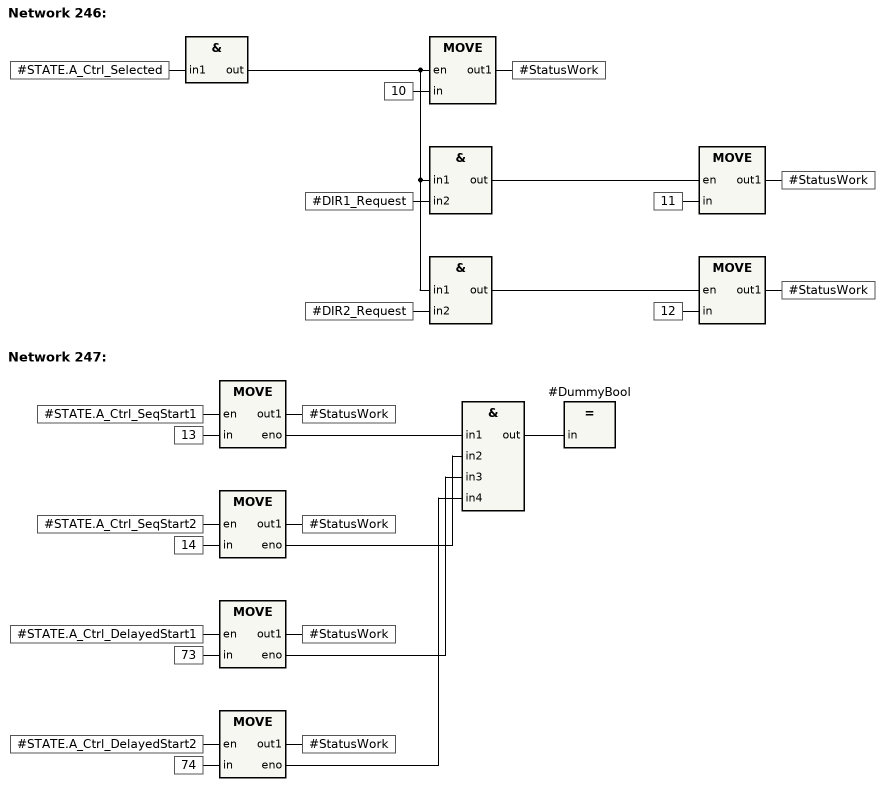
   IF #STATE.A_Ctrl_Selected THEN #StatusWork := 10; END_IF;
   IF #STATE.A_Ctrl_Selected AND #DIR1_Request THEN #StatusWork := 11; END_IF;
   IF #STATE.A_Ctrl_Selected AND #DIR2_Request THEN #StatusWork := 12; END_IF;
END_REGION

REGION Network 247
   // ENO of a box is taken as its EN; it also drops when the box reports an error
   IF #STATE.A_Ctrl_SeqStart1 THEN #StatusWork := 13; END_IF;
   IF #STATE.A_Ctrl_SeqStart2 THEN #StatusWork := 14; END_IF;
   IF #STATE.A_Ctrl_DelayedStart1 THEN #StatusWork := 73; END_IF;
   IF #STATE.A_Ctrl_DelayedStart2 THEN #StatusWork := 74; END_IF;
   #DummyBool := #STATE.A_Ctrl_SeqStart1 AND #STATE.A_Ctrl_SeqStart2 AND #STATE.A_Ctrl_DelayedStart1 AND #STATE.A_Ctrl_DelayedStart2;
END_REGION

REGION Network 248
   // Build 008 - 30.09.2020 (EXTBOB):  State Alarm Neg added to avoid start warn in case of alarm state
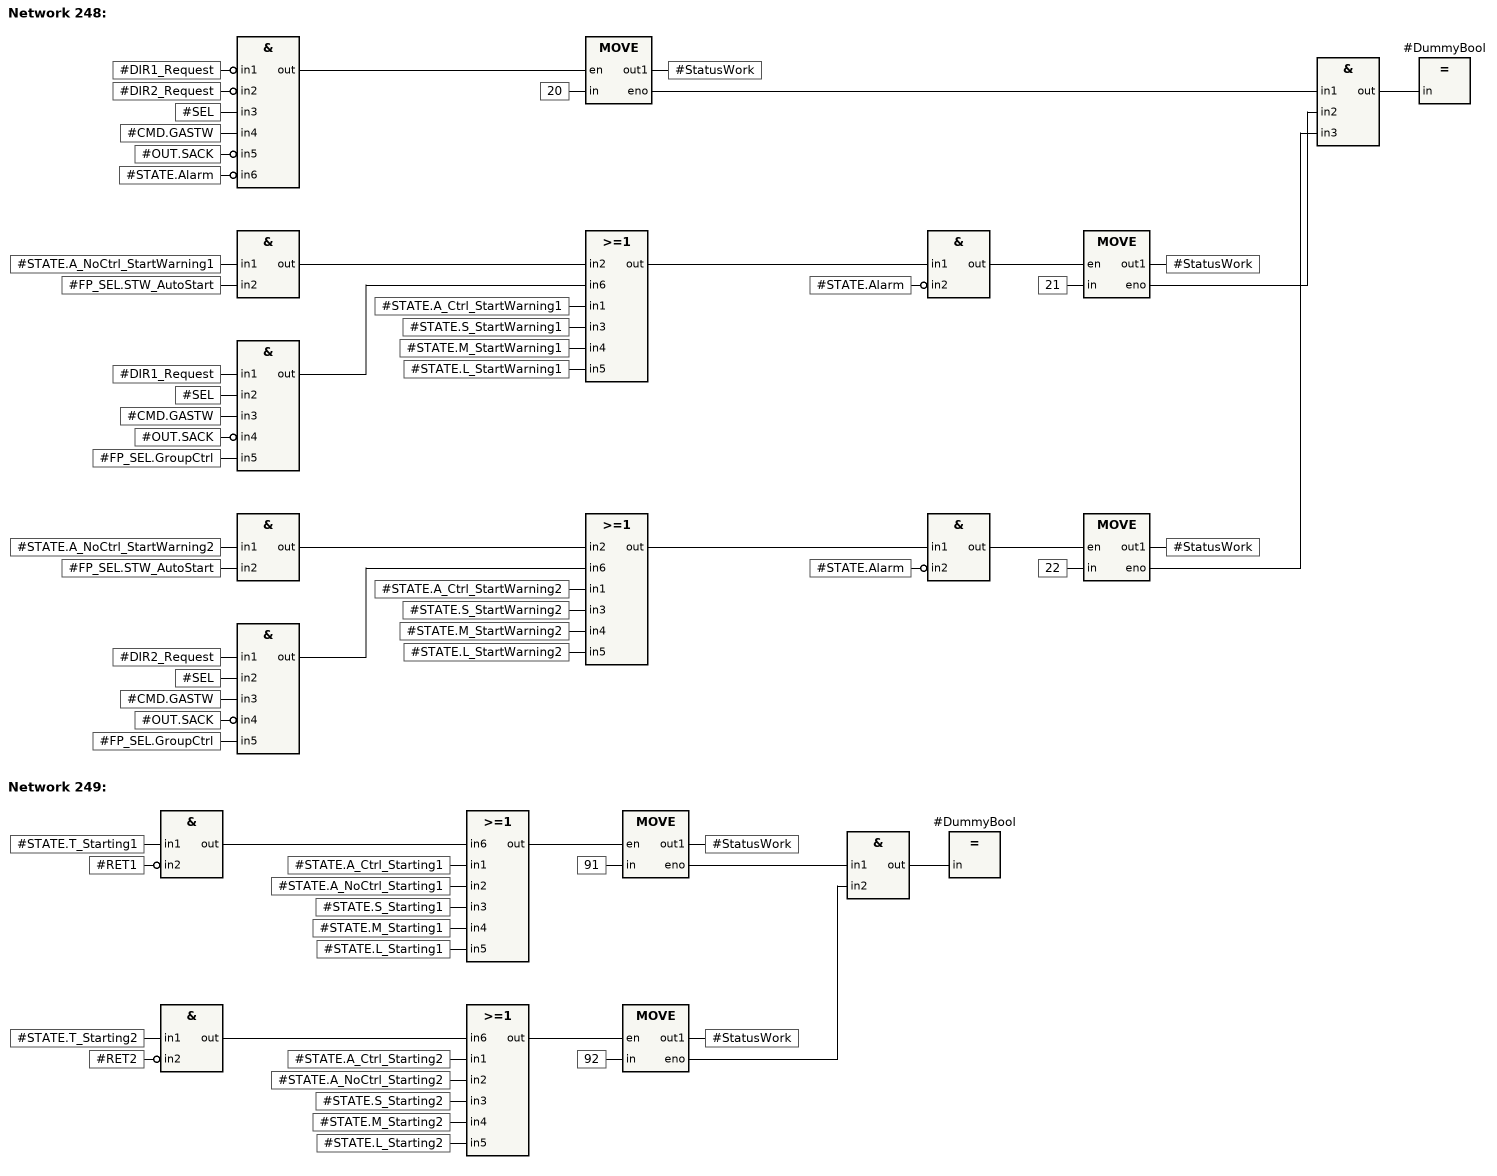
   // ENO of a box is taken as its EN; it also drops when the box reports an error
   #_w1 := NOT #DIR1_Request AND NOT #DIR2_Request AND #SEL AND #CMD.GASTW AND NOT #OUT.SACK AND NOT #STATE.Alarm;
   IF #_w1 THEN #StatusWork := 20; END_IF;
   #_w2 := ((#STATE.A_NoCtrl_StartWarning1 AND #FP_SEL.STW_AutoStart) OR (#DIR1_Request AND #SEL AND #CMD.GASTW AND NOT #OUT.SACK AND #FP_SEL.GroupCtrl) OR #STATE.A_Ctrl_StartWarning1 OR #STATE.S_StartWarning1 OR #STATE.M_StartWarning1 OR #STATE.L_StartWarning1) AND NOT #STATE.Alarm;
   IF #_w2 THEN #StatusWork := 21; END_IF;
   #_w3 := ((#STATE.A_NoCtrl_StartWarning2 AND #FP_SEL.STW_AutoStart) OR (#DIR2_Request AND #SEL AND #CMD.GASTW AND NOT #OUT.SACK AND #FP_SEL.GroupCtrl) OR #STATE.A_Ctrl_StartWarning2 OR #STATE.S_StartWarning2 OR #STATE.M_StartWarning2 OR #STATE.L_StartWarning2) AND NOT #STATE.Alarm;
   IF #_w3 THEN #StatusWork := 22; END_IF;
   #DummyBool := #_w1 AND #_w2 AND #_w3;
END_REGION

REGION Network 249
   // ENO of a box is taken as its EN; it also drops when the box reports an error
   #_w1 := (#STATE.T_Starting1 AND NOT #RET1) OR #STATE.A_Ctrl_Starting1 OR #STATE.A_NoCtrl_Starting1 OR #STATE.S_Starting1 OR #STATE.M_Starting1 OR #STATE.L_Starting1;
   IF #_w1 THEN #StatusWork := 91; END_IF;
   #_w2 := (#STATE.T_Starting2 AND NOT #RET2) OR #STATE.A_Ctrl_Starting2 OR #STATE.A_NoCtrl_Starting2 OR #STATE.S_Starting2 OR #STATE.M_Starting2 OR #STATE.L_Starting2;
   IF #_w2 THEN #StatusWork := 92; END_IF;
   #DummyBool := #_w1 AND #_w2;
END_REGION

REGION Network 250
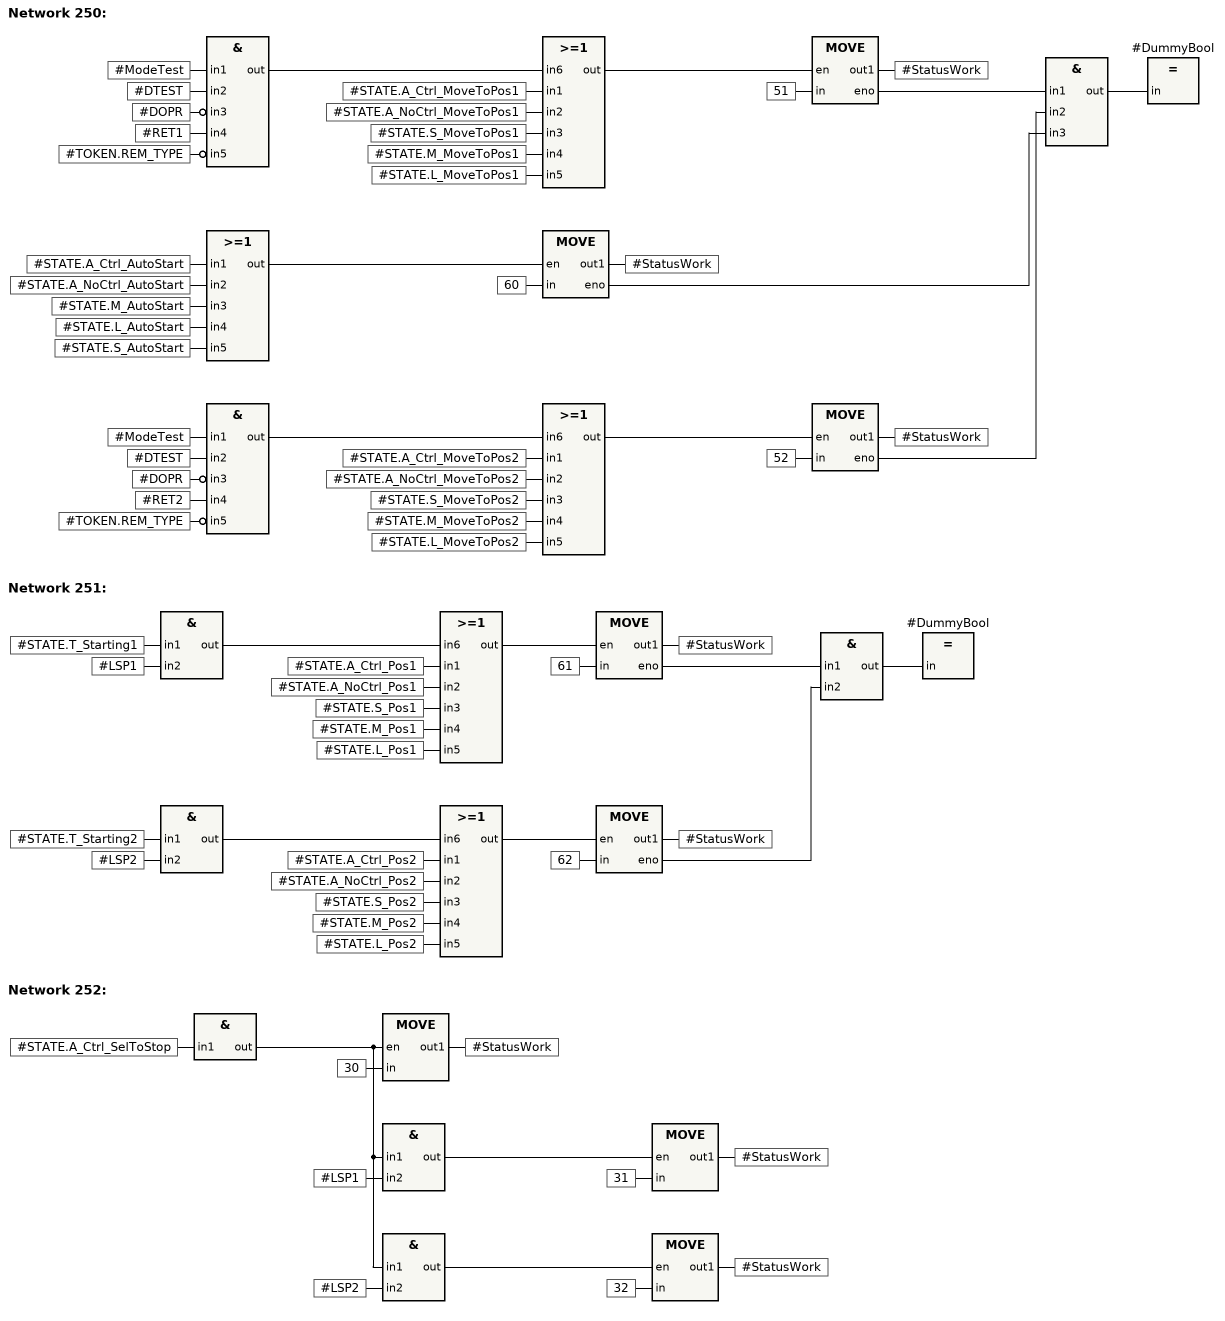
   // ENO of a box is taken as its EN; it also drops when the box reports an error
   #_w1 := (#ModeTest AND #DTEST AND NOT #DOPR AND #RET1 AND NOT #TOKEN.REM_TYPE) OR #STATE.A_Ctrl_MoveToPos1 OR #STATE.A_NoCtrl_MoveToPos1 OR #STATE.S_MoveToPos1 OR #STATE.M_MoveToPos1 OR #STATE.L_MoveToPos1;
   IF #_w1 THEN #StatusWork := 51; END_IF;
   #_w2 := (#ModeTest AND #DTEST AND NOT #DOPR AND #RET2 AND NOT #TOKEN.REM_TYPE) OR #STATE.A_Ctrl_MoveToPos2 OR #STATE.A_NoCtrl_MoveToPos2 OR #STATE.S_MoveToPos2 OR #STATE.M_MoveToPos2 OR #STATE.L_MoveToPos2;
   IF #_w2 THEN #StatusWork := 52; END_IF;
   #_w3 := #STATE.A_Ctrl_AutoStart OR #STATE.A_NoCtrl_AutoStart OR #STATE.M_AutoStart OR #STATE.L_AutoStart OR #STATE.S_AutoStart;
   IF #_w3 THEN #StatusWork := 60; END_IF;
   #DummyBool := #_w1 AND #_w2 AND #_w3;
END_REGION

REGION Network 251
   // ENO of a box is taken as its EN; it also drops when the box reports an error
   #_w1 := (#STATE.T_Starting1 AND #LSP1) OR #STATE.A_Ctrl_Pos1 OR #STATE.A_NoCtrl_Pos1 OR #STATE.S_Pos1 OR #STATE.M_Pos1 OR #STATE.L_Pos1;
   IF #_w1 THEN #StatusWork := 61; END_IF;
   #_w2 := (#STATE.T_Starting2 AND #LSP2) OR #STATE.A_Ctrl_Pos2 OR #STATE.A_NoCtrl_Pos2 OR #STATE.S_Pos2 OR #STATE.M_Pos2 OR #STATE.L_Pos2;
   IF #_w2 THEN #StatusWork := 62; END_IF;
   #DummyBool := #_w1 AND #_w2;
END_REGION

REGION Network 252
   IF #STATE.A_Ctrl_SelToStop THEN #StatusWork := 30; END_IF;
   IF #STATE.A_Ctrl_SelToStop AND #LSP1 THEN #StatusWork := 31; END_IF;
   IF #STATE.A_Ctrl_SelToStop AND #LSP2 THEN #StatusWork := 32; END_IF;
END_REGION

REGION Network 253
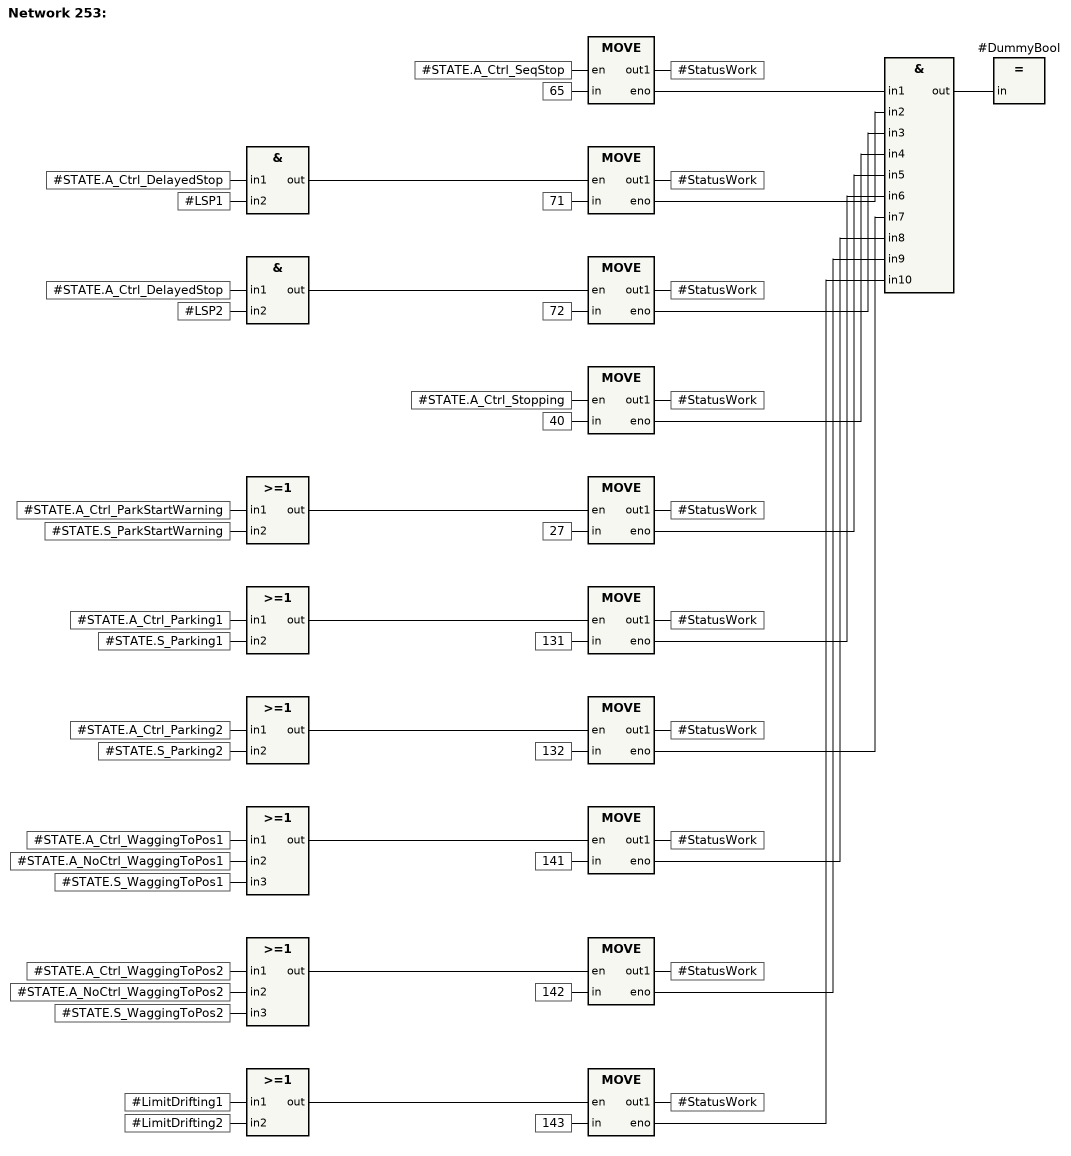
   // ENO of a box is taken as its EN; it also drops when the box reports an error
   IF #STATE.A_Ctrl_SeqStop THEN #StatusWork := 65; END_IF;
   #_w1 := #STATE.A_Ctrl_DelayedStop AND #LSP1;
   IF #_w1 THEN #StatusWork := 71; END_IF;
   #_w2 := #STATE.A_Ctrl_DelayedStop AND #LSP2;
   IF #_w2 THEN #StatusWork := 72; END_IF;
   IF #STATE.A_Ctrl_Stopping THEN #StatusWork := 40; END_IF;
   #_w3 := #STATE.A_Ctrl_ParkStartWarning OR #STATE.S_ParkStartWarning;
   IF #_w3 THEN #StatusWork := 27; END_IF;
   #_w4 := #STATE.A_Ctrl_Parking1 OR #STATE.S_Parking1;
   IF #_w4 THEN #StatusWork := 131; END_IF;
   #_w5 := #STATE.A_Ctrl_Parking2 OR #STATE.S_Parking2;
   IF #_w5 THEN #StatusWork := 132; END_IF;
   #_w6 := #STATE.A_Ctrl_WaggingToPos1 OR #STATE.A_NoCtrl_WaggingToPos1 OR #STATE.S_WaggingToPos1;
   IF #_w6 THEN #StatusWork := 141; END_IF;
   #_w7 := #STATE.A_Ctrl_WaggingToPos2 OR #STATE.A_NoCtrl_WaggingToPos2 OR #STATE.S_WaggingToPos2;
   IF #_w7 THEN #StatusWork := 142; END_IF;
   #_w8 := #LimitDrifting1 OR #LimitDrifting2;
   IF #_w8 THEN #StatusWork := 143; END_IF;
   #DummyBool := #STATE.A_Ctrl_SeqStop AND #_w1 AND #_w2 AND #STATE.A_Ctrl_Stopping AND #_w3 AND #_w4 AND #_w5 AND #_w6 AND #_w7 AND #_w8;
END_REGION

REGION Network 254
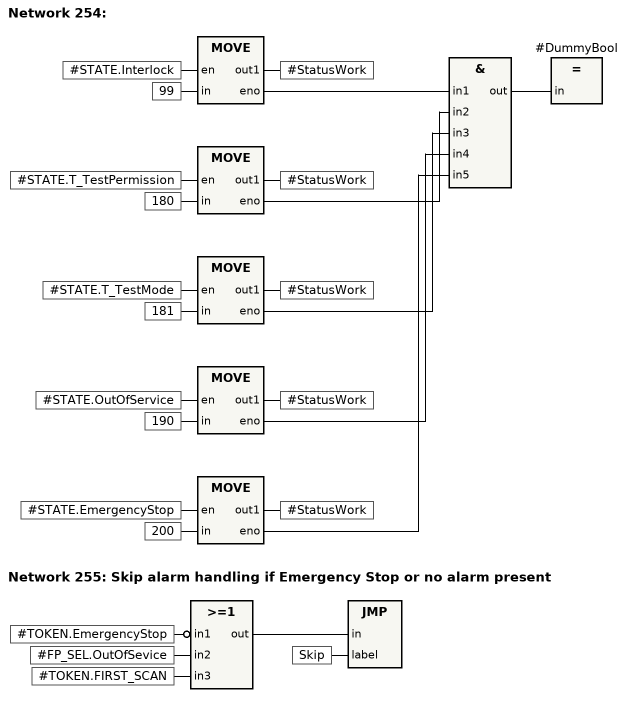
   // ENO of a box is taken as its EN; it also drops when the box reports an error
   IF #STATE.Interlock THEN #StatusWork := 99; END_IF;
   IF #STATE.T_TestPermission THEN #StatusWork := 180; END_IF;
   IF #STATE.T_TestMode THEN #StatusWork := 181; END_IF;
   IF #STATE.OutOfService THEN #StatusWork := 190; END_IF;
   IF #STATE.EmergencyStop THEN #StatusWork := 200; END_IF;
   #DummyBool := #STATE.Interlock AND #STATE.T_TestPermission AND #STATE.T_TestMode AND #STATE.OutOfService AND #STATE.EmergencyStop;
END_REGION

REGION Network 255: Skip alarm handling if Emergency Stop or no alarm present
   IF NOT #TOKEN.EmergencyStop OR #FP_SEL.OutOfSevice OR #TOKEN.FIRST_SCAN THEN GOTO Skip; END_IF;
END_REGION

REGION Network 256: Alarm Present
   // Build 006 - 28 Jan 2020 (EXTBOB) : Torque fault also considered  in Local 
   // &Manual Mode startwarning time, OK Alarm used in place of ALARM_AlarmPresent 
   // and removed TestMode
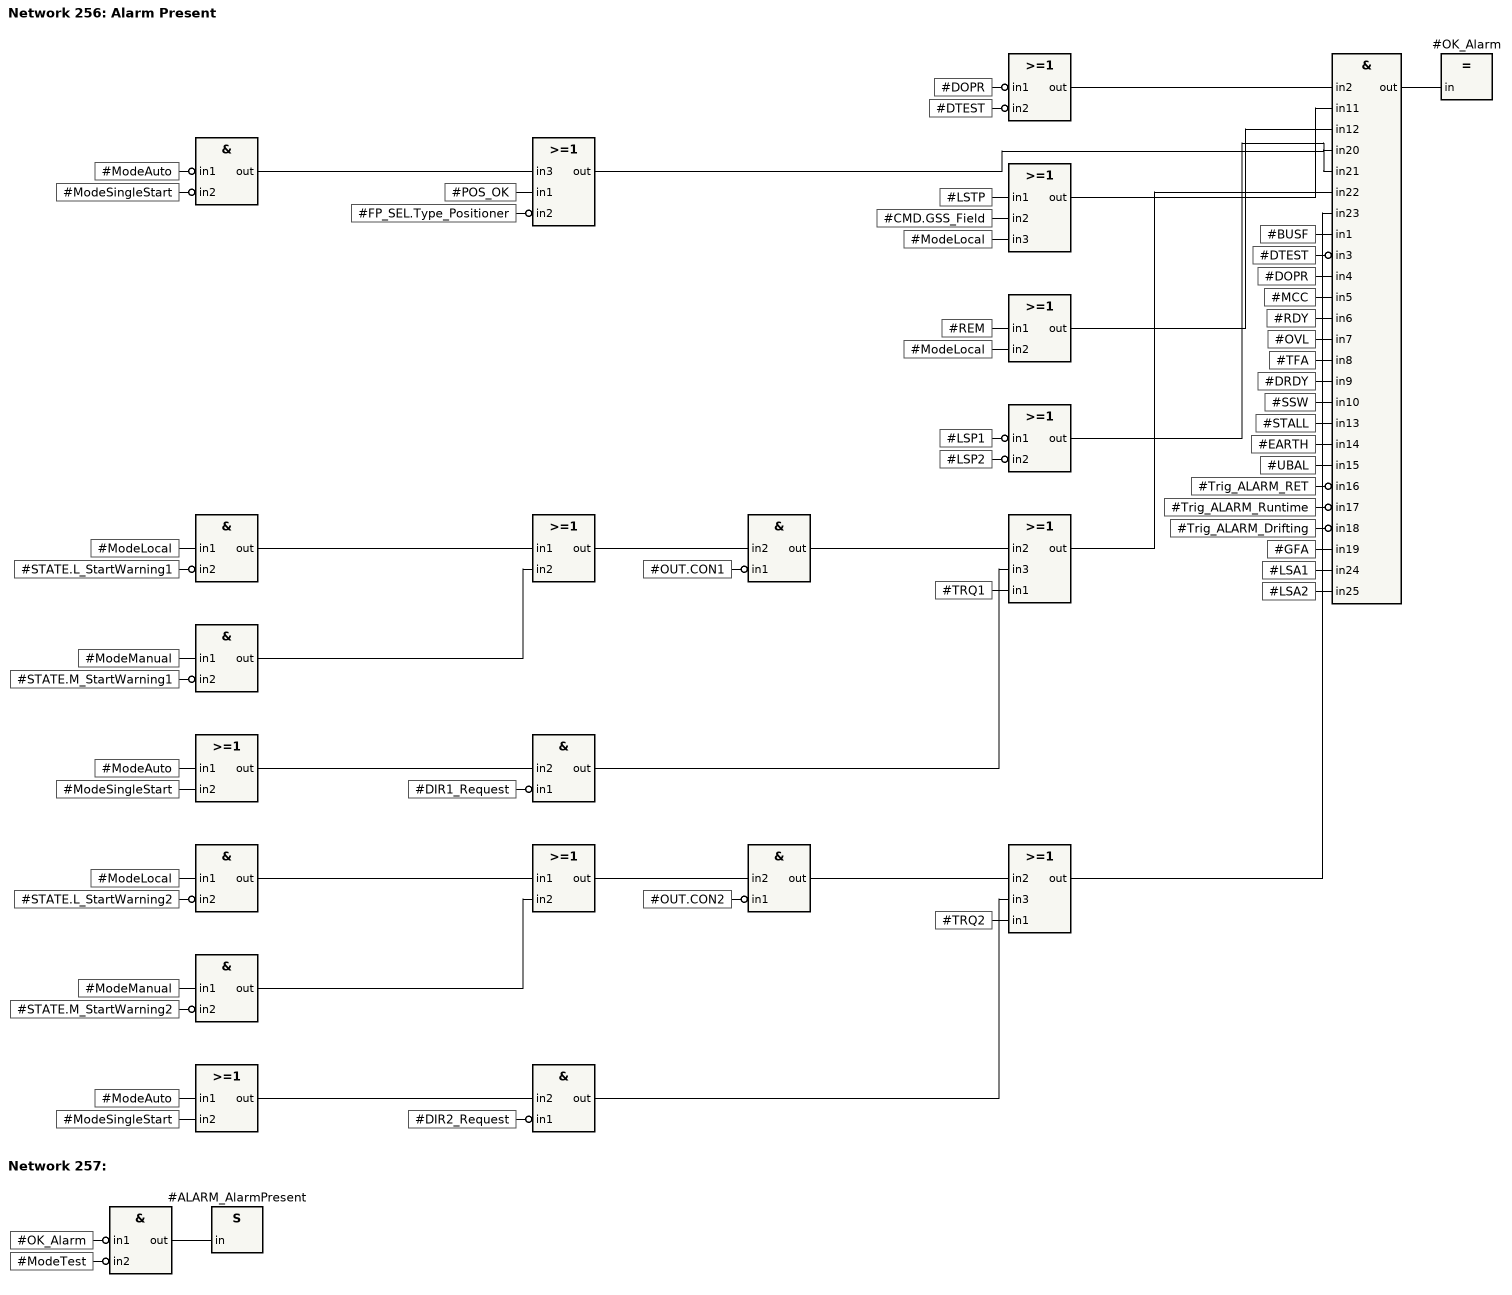
   #OK_Alarm := (NOT #DOPR OR NOT #DTEST) AND (#LSTP OR #CMD.GSS_Field OR #ModeLocal) AND (#REM OR #ModeLocal) AND (NOT #LSP1 OR NOT #LSP2) AND ((NOT #ModeAuto AND NOT #ModeSingleStart) OR #POS_OK OR NOT #FP_SEL.Type_Positioner) AND ((((#ModeLocal AND NOT #STATE.L_StartWarning1) OR (#ModeManual AND NOT #STATE.M_StartWarning1)) AND NOT #OUT.CON1) OR ((#ModeAuto OR #ModeSingleStart) AND NOT #DIR1_Request) OR #TRQ1) AND ((((#ModeLocal AND NOT #STATE.L_StartWarning2) OR (#ModeManual AND NOT #STATE.M_StartWarning2)) AND NOT #OUT.CON2) OR ((#ModeAuto OR #ModeSingleStart) AND NOT #DIR2_Request) OR #TRQ2) AND #BUSF AND NOT #DTEST AND #DOPR AND #MCC AND #RDY AND #OVL AND #TFA AND #DRDY AND #SSW AND #STALL AND #EARTH AND #UBAL AND NOT #Trig_ALARM_RET AND NOT #Trig_ALARM_Runtime AND NOT #Trig_ALARM_Drifting AND #GFA AND #LSA1 AND #LSA2;
END_REGION

REGION Network 257
   // Build 006 - 28 Jan 2020 (EXTBOB) : Newly added to make this logic same as other PLC brands
   IF NOT #OK_Alarm AND NOT #ModeTest THEN #ALARM_AlarmPresent := TRUE; END_IF;
END_REGION

REGION Network 258
   // Build 006 - 28 Jan 2020 (EXTBOB) : Newly added to make this logic same as other PLC brands
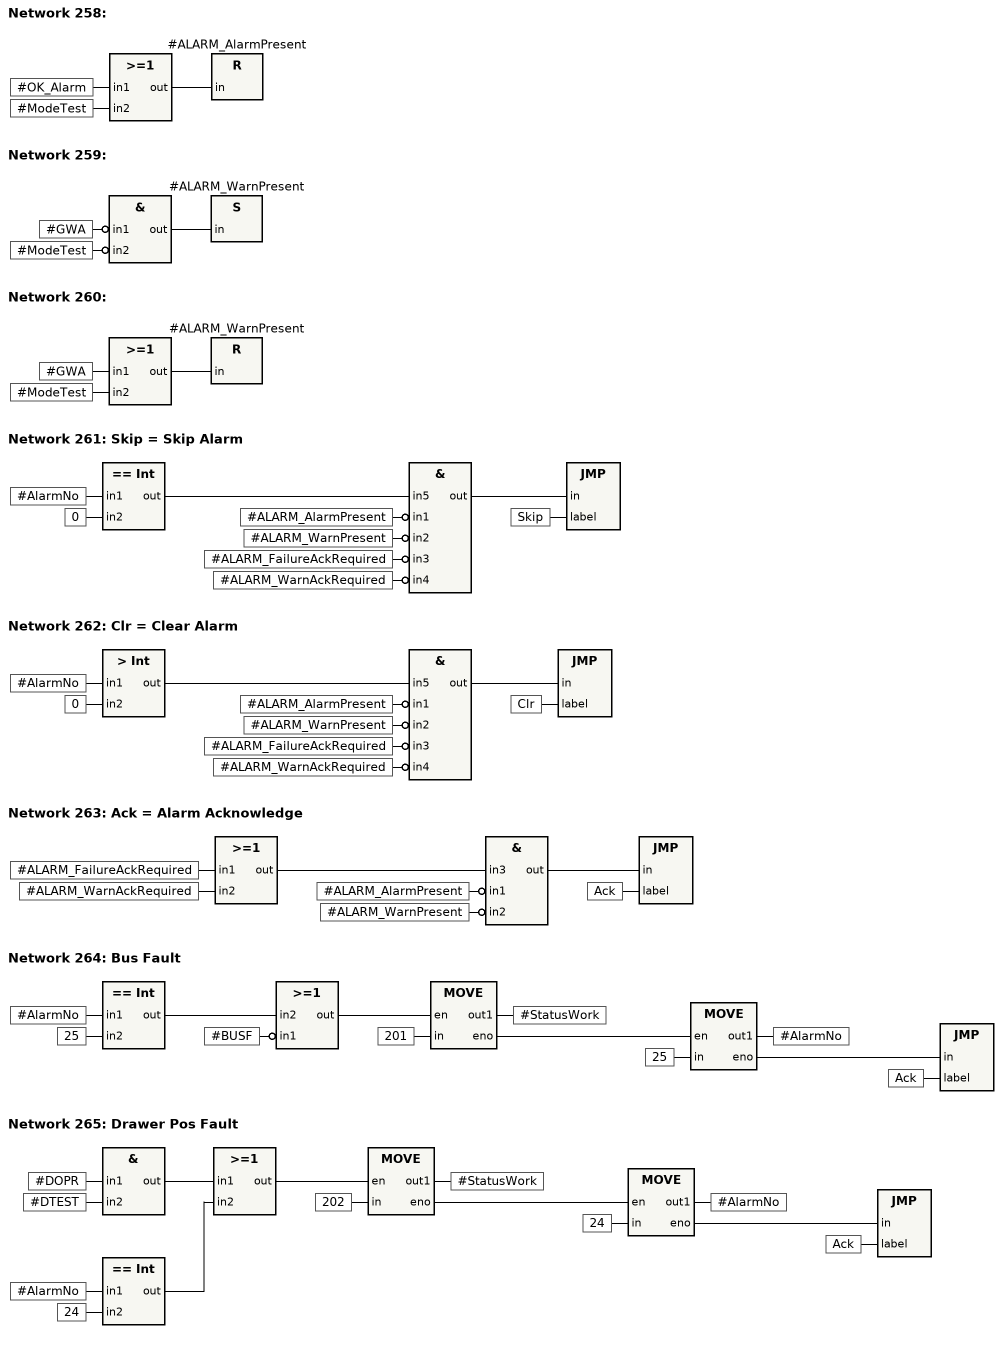
   IF #OK_Alarm OR #ModeTest THEN #ALARM_AlarmPresent := FALSE; END_IF;
END_REGION

REGION Network 259
   // Build 006 - 28 Jan 2020 (EXTBOB) : Newly added to make this logic same as other PLC brands - Modified the existing logic of ALARM_WarnPresent
   IF NOT #GWA AND NOT #ModeTest THEN #ALARM_WarnPresent := TRUE; END_IF;
END_REGION

REGION Network 260
   // Build 006 - 28 Jan 2020 (EXTBOB) : Newly added to make this logic same as other PLC brands
   IF #GWA OR #ModeTest THEN #ALARM_WarnPresent := FALSE; END_IF;
END_REGION

REGION Network 261: Skip = Skip Alarm
   IF (#AlarmNo = 0) AND NOT #ALARM_AlarmPresent AND NOT #ALARM_WarnPresent AND NOT #ALARM_FailureAckRequired AND NOT #ALARM_WarnAckRequired THEN
       GOTO Skip;
   END_IF;
END_REGION

REGION Network 262: Clr = Clear Alarm
   IF (#AlarmNo > 0) AND NOT #ALARM_AlarmPresent AND NOT #ALARM_WarnPresent AND NOT #ALARM_FailureAckRequired AND NOT #ALARM_WarnAckRequired THEN
       GOTO Clr;
   END_IF;
END_REGION

REGION Network 263: Ack = Alarm Acknowledge
   IF (#ALARM_FailureAckRequired OR #ALARM_WarnAckRequired) AND NOT #ALARM_AlarmPresent AND NOT #ALARM_WarnPresent THEN
       GOTO Ack;
   END_IF;
END_REGION

REGION Network 264: Bus Fault
   // ENO of a box is taken as its EN; it also drops when the box reports an error
   #_w1 := (#AlarmNo = 25) OR NOT #BUSF;
   IF #_w1 THEN
       #StatusWork := 201;
       #AlarmNo := 25;
       GOTO Ack;
   END_IF;
END_REGION

REGION Network 265: Drawer Pos Fault
   // ENO of a box is taken as its EN; it also drops when the box reports an error
   #_w1 := (#DOPR AND #DTEST) OR (#AlarmNo = 24);
   IF #_w1 THEN
       #StatusWork := 202;
       #AlarmNo := 24;
       GOTO Ack;
   END_IF;
END_REGION

REGION Network 266: Drawer Not In Operation Pos
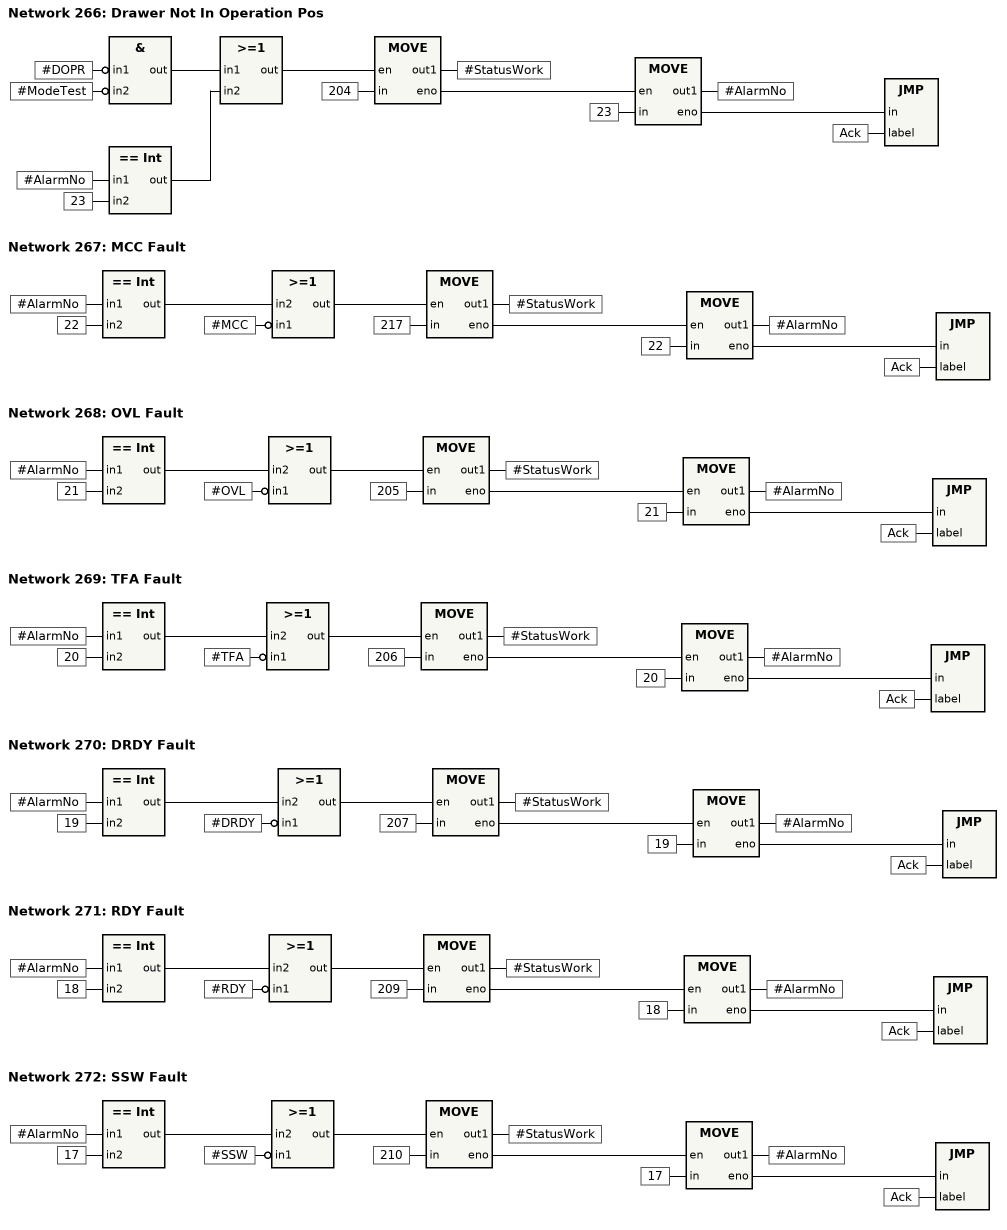
   // ENO of a box is taken as its EN; it also drops when the box reports an error
   #_w1 := (NOT #DOPR AND NOT #ModeTest) OR (#AlarmNo = 23);
   IF #_w1 THEN
       #StatusWork := 204;
       #AlarmNo := 23;
       GOTO Ack;
   END_IF;
END_REGION

REGION Network 267: MCC Fault
   // ENO of a box is taken as its EN; it also drops when the box reports an error
   #_w1 := (#AlarmNo = 22) OR NOT #MCC;
   IF #_w1 THEN
       #StatusWork := 217;
       #AlarmNo := 22;
       GOTO Ack;
   END_IF;
END_REGION

REGION Network 268: OVL Fault
   // ENO of a box is taken as its EN; it also drops when the box reports an error
   #_w1 := (#AlarmNo = 21) OR NOT #OVL;
   IF #_w1 THEN
       #StatusWork := 205;
       #AlarmNo := 21;
       GOTO Ack;
   END_IF;
END_REGION

REGION Network 269: TFA Fault
   // ENO of a box is taken as its EN; it also drops when the box reports an error
   #_w1 := (#AlarmNo = 20) OR NOT #TFA;
   IF #_w1 THEN
       #StatusWork := 206;
       #AlarmNo := 20;
       GOTO Ack;
   END_IF;
END_REGION

REGION Network 270: DRDY Fault
   // ENO of a box is taken as its EN; it also drops when the box reports an error
   #_w1 := (#AlarmNo = 19) OR NOT #DRDY;
   IF #_w1 THEN
       #StatusWork := 207;
       #AlarmNo := 19;
       GOTO Ack;
   END_IF;
END_REGION

REGION Network 271: RDY Fault
   // ENO of a box is taken as its EN; it also drops when the box reports an error
   #_w1 := (#AlarmNo = 18) OR NOT #RDY;
   IF #_w1 THEN
       #StatusWork := 209;
       #AlarmNo := 18;
       GOTO Ack;
   END_IF;
END_REGION

REGION Network 272: SSW Fault
   // ENO of a box is taken as its EN; it also drops when the box reports an error
   #_w1 := (#AlarmNo = 17) OR NOT #SSW;
   IF #_w1 THEN
       #StatusWork := 210;
       #AlarmNo := 17;
       GOTO Ack;
   END_IF;
END_REGION

REGION Network 273: LSTP Fault
